   // UNICODE_TO_GBK[27326] := 16#8092;
   // UNICODE_TO_GBK[27327] := 16#C34B;
   // UNICODE_TO_GBK[27328] := 16#8093;
   // UNICODE_TO_GBK[27329] := 16#EBC1;
   // UNICODE_TO_GBK[27330] := 16#8094;
   // UNICODE_TO_GBK[27331] := 16#C34C;
   // UNICODE_TO_GBK[27332] := 16#8095;
   // UNICODE_TO_GBK[27333] := 16#C34D;
   // UNICODE_TO_GBK[27334] := 16#8096;
   // UNICODE_TO_GBK[27335] := 16#D0A4;
   // UNICODE_TO_GBK[27336] := 16#8097;
   // UNICODE_TO_GBK[27337] := 16#C34E;
   // UNICODE_TO_GBK[27338] := 16#8098;
   // UNICODE_TO_GBK[27339] := 16#D6E2;
   // UNICODE_TO_GBK[27340] := 16#8099;
   // UNICODE_TO_GBK[27341] := 16#C34F;
   // UNICODE_TO_GBK[27342] := 16#809A;
   // UNICODE_TO_GBK[27343] := 16#B6C7;
   // UNICODE_TO_GBK[27344] := 16#809B;
   // UNICODE_TO_GBK[27345] := 16#B8D8;
   // UNICODE_TO_GBK[27346] := 16#809C;
   // UNICODE_TO_GBK[27347] := 16#EBC0;
   // UNICODE_TO_GBK[27348] := 16#809D;
   // UNICODE_TO_GBK[27349] := 16#B8CE;
   // UNICODE_TO_GBK[27350] := 16#809E;
   // UNICODE_TO_GBK[27351] := 16#C350;
   // UNICODE_TO_GBK[27352] := 16#809F;
   // UNICODE_TO_GBK[27353] := 16#EBBF;
   // UNICODE_TO_GBK[27354] := 16#80A0;
   // UNICODE_TO_GBK[27355] := 16#B3A6;
   // UNICODE_TO_GBK[27356] := 16#80A1;
   // UNICODE_TO_GBK[27357] := 16#B9C9;
   // UNICODE_TO_GBK[27358] := 16#80A2;
   // UNICODE_TO_GBK[27359] := 16#D6AB;
   // UNICODE_TO_GBK[27360] := 16#80A3;
   // UNICODE_TO_GBK[27361] := 16#C351;
   // UNICODE_TO_GBK[27362] := 16#80A4;
   // UNICODE_TO_GBK[27363] := 16#B7F4;
   // UNICODE_TO_GBK[27364] := 16#80A5;
   // UNICODE_TO_GBK[27365] := 16#B7CA;
   // UNICODE_TO_GBK[27366] := 16#80A6;
   // UNICODE_TO_GBK[27367] := 16#C352;
   // UNICODE_TO_GBK[27368] := 16#80A7;
   // UNICODE_TO_GBK[27369] := 16#C353;
   // UNICODE_TO_GBK[27370] := 16#80A8;
   // UNICODE_TO_GBK[27371] := 16#C354;
   // UNICODE_TO_GBK[27372] := 16#80A9;
   // UNICODE_TO_GBK[27373] := 16#BCE7;
   // UNICODE_TO_GBK[27374] := 16#80AA;
   // UNICODE_TO_GBK[27375] := 16#B7BE;
   // UNICODE_TO_GBK[27376] := 16#80AB;
   // UNICODE_TO_GBK[27377] := 16#EBC6;
   // UNICODE_TO_GBK[27378] := 16#80AC;
   // UNICODE_TO_GBK[27379] := 16#C355;
   // UNICODE_TO_GBK[27380] := 16#80AD;
   // UNICODE_TO_GBK[27381] := 16#EBC7;
   // UNICODE_TO_GBK[27382] := 16#80AE;
   // UNICODE_TO_GBK[27383] := 16#B0B9;
   // UNICODE_TO_GBK[27384] := 16#80AF;
   // UNICODE_TO_GBK[27385] := 16#BFCF;
   // UNICODE_TO_GBK[27386] := 16#80B0;
   // UNICODE_TO_GBK[27387] := 16#C356;
   // UNICODE_TO_GBK[27388] := 16#80B1;
   // UNICODE_TO_GBK[27389] := 16#EBC5;
   // UNICODE_TO_GBK[27390] := 16#80B2;
   // UNICODE_TO_GBK[27391] := 16#D3FD;
   // UNICODE_TO_GBK[27392] := 16#80B3;
   // UNICODE_TO_GBK[27393] := 16#C357;
   // UNICODE_TO_GBK[27394] := 16#80B4;
   // UNICODE_TO_GBK[27395] := 16#EBC8;
   // UNICODE_TO_GBK[27396] := 16#80B5;
   // UNICODE_TO_GBK[27397] := 16#C358;
   // UNICODE_TO_GBK[27398] := 16#80B6;
   // UNICODE_TO_GBK[27399] := 16#C359;
   // UNICODE_TO_GBK[27400] := 16#80B7;
   // UNICODE_TO_GBK[27401] := 16#EBC9;
   // UNICODE_TO_GBK[27402] := 16#80B8;
   // UNICODE_TO_GBK[27403] := 16#C35A;
   // UNICODE_TO_GBK[27404] := 16#80B9;
   // UNICODE_TO_GBK[27405] := 16#C35B;
   // UNICODE_TO_GBK[27406] := 16#80BA;
   // UNICODE_TO_GBK[27407] := 16#B7CE;
   // UNICODE_TO_GBK[27408] := 16#80BB;
   // UNICODE_TO_GBK[27409] := 16#C35C;
   // UNICODE_TO_GBK[27410] := 16#80BC;
   // UNICODE_TO_GBK[27411] := 16#EBC2;
   // UNICODE_TO_GBK[27412] := 16#80BD;
   // UNICODE_TO_GBK[27413] := 16#EBC4;
   // UNICODE_TO_GBK[27414] := 16#80BE;
   // UNICODE_TO_GBK[27415] := 16#C9F6;
   // UNICODE_TO_GBK[27416] := 16#80BF;
   // UNICODE_TO_GBK[27417] := 16#D6D7;
   // UNICODE_TO_GBK[27418] := 16#80C0;
   // UNICODE_TO_GBK[27419] := 16#D5CD;
   // UNICODE_TO_GBK[27420] := 16#80C1;
   // UNICODE_TO_GBK[27421] := 16#D0B2;
   // UNICODE_TO_GBK[27422] := 16#80C2;
   // UNICODE_TO_GBK[27423] := 16#EBCF;
   // UNICODE_TO_GBK[27424] := 16#80C3;
   // UNICODE_TO_GBK[27425] := 16#CEB8;
   // UNICODE_TO_GBK[27426] := 16#80C4;
   // UNICODE_TO_GBK[27427] := 16#EBD0;
   // UNICODE_TO_GBK[27428] := 16#80C5;
   // UNICODE_TO_GBK[27429] := 16#C35D;
   // UNICODE_TO_GBK[27430] := 16#80C6;
   // UNICODE_TO_GBK[27431] := 16#B5A8;
   // UNICODE_TO_GBK[27432] := 16#80C7;
   // UNICODE_TO_GBK[27433] := 16#C35E;
   // UNICODE_TO_GBK[27434] := 16#80C8;
   // UNICODE_TO_GBK[27435] := 16#C35F;
   // UNICODE_TO_GBK[27436] := 16#80C9;
   // UNICODE_TO_GBK[27437] := 16#C360;
   // UNICODE_TO_GBK[27438] := 16#80CA;
   // UNICODE_TO_GBK[27439] := 16#C361;
   // UNICODE_TO_GBK[27440] := 16#80CB;
   // UNICODE_TO_GBK[27441] := 16#C362;
   // UNICODE_TO_GBK[27442] := 16#80CC;
   // UNICODE_TO_GBK[27443] := 16#B1B3;
   // UNICODE_TO_GBK[27444] := 16#80CD;
   // UNICODE_TO_GBK[27445] := 16#EBD2;
   // UNICODE_TO_GBK[27446] := 16#80CE;
   // UNICODE_TO_GBK[27447] := 16#CCA5;
   // UNICODE_TO_GBK[27448] := 16#80CF;
   // UNICODE_TO_GBK[27449] := 16#C363;
   // UNICODE_TO_GBK[27450] := 16#80D0;
   // UNICODE_TO_GBK[27451] := 16#C364;
   // UNICODE_TO_GBK[27452] := 16#80D1;
   // UNICODE_TO_GBK[27453] := 16#C365;
   // UNICODE_TO_GBK[27454] := 16#80D2;
   // UNICODE_TO_GBK[27455] := 16#C366;
   // UNICODE_TO_GBK[27456] := 16#80D3;
   // UNICODE_TO_GBK[27457] := 16#C367;
   // UNICODE_TO_GBK[27458] := 16#80D4;
   // UNICODE_TO_GBK[27459] := 16#C368;
   // UNICODE_TO_GBK[27460] := 16#80D5;
   // UNICODE_TO_GBK[27461] := 16#C369;
   // UNICODE_TO_GBK[27462] := 16#80D6;
   // UNICODE_TO_GBK[27463] := 16#C5D6;
   // UNICODE_TO_GBK[27464] := 16#80D7;
   // UNICODE_TO_GBK[27465] := 16#EBD3;
   // UNICODE_TO_GBK[27466] := 16#80D8;
   // UNICODE_TO_GBK[27467] := 16#C36A;
   // UNICODE_TO_GBK[27468] := 16#80D9;
   // UNICODE_TO_GBK[27469] := 16#EBD1;
   // UNICODE_TO_GBK[27470] := 16#80DA;
   // UNICODE_TO_GBK[27471] := 16#C5DF;
   // UNICODE_TO_GBK[27472] := 16#80DB;
   // UNICODE_TO_GBK[27473] := 16#EBCE;
   // UNICODE_TO_GBK[27474] := 16#80DC;
   // UNICODE_TO_GBK[27475] := 16#CAA4;
   // UNICODE_TO_GBK[27476] := 16#80DD;
   // UNICODE_TO_GBK[27477] := 16#EBD5;
   // UNICODE_TO_GBK[27478] := 16#80DE;
   // UNICODE_TO_GBK[27479] := 16#B0FB;
   // UNICODE_TO_GBK[27480] := 16#80DF;
   // UNICODE_TO_GBK[27481] := 16#C36B;
   // UNICODE_TO_GBK[27482] := 16#80E0;
   // UNICODE_TO_GBK[27483] := 16#C36C;
   // UNICODE_TO_GBK[27484] := 16#80E1;
   // UNICODE_TO_GBK[27485] := 16#BAFA;
   // UNICODE_TO_GBK[27486] := 16#80E2;
   // UNICODE_TO_GBK[27487] := 16#C36D;
   // UNICODE_TO_GBK[27488] := 16#80E3;
   // UNICODE_TO_GBK[27489] := 16#C36E;
   // UNICODE_TO_GBK[27490] := 16#80E4;
   // UNICODE_TO_GBK[27491] := 16#D8B7;
   // UNICODE_TO_GBK[27492] := 16#80E5;
   // UNICODE_TO_GBK[27493] := 16#F1E3;
   // UNICODE_TO_GBK[27494] := 16#80E6;
   // UNICODE_TO_GBK[27495] := 16#C36F;
   // UNICODE_TO_GBK[27496] := 16#80E7;
   // UNICODE_TO_GBK[27497] := 16#EBCA;
   // UNICODE_TO_GBK[27498] := 16#80E8;
   // UNICODE_TO_GBK[27499] := 16#EBCB;
   // UNICODE_TO_GBK[27500] := 16#80E9;
   // UNICODE_TO_GBK[27501] := 16#EBCC;
   // UNICODE_TO_GBK[27502] := 16#80EA;
   // UNICODE_TO_GBK[27503] := 16#EBCD;
   // UNICODE_TO_GBK[27504] := 16#80EB;
   // UNICODE_TO_GBK[27505] := 16#EBD6;
   // UNICODE_TO_GBK[27506] := 16#80EC;
   // UNICODE_TO_GBK[27507] := 16#E6C0;
   // UNICODE_TO_GBK[27508] := 16#80ED;
   // UNICODE_TO_GBK[27509] := 16#EBD9;
   // UNICODE_TO_GBK[27510] := 16#80EE;
   // UNICODE_TO_GBK[27511] := 16#C370;
   // UNICODE_TO_GBK[27512] := 16#80EF;
   // UNICODE_TO_GBK[27513] := 16#BFE8;
   // UNICODE_TO_GBK[27514] := 16#80F0;
   // UNICODE_TO_GBK[27515] := 16#D2C8;
   // UNICODE_TO_GBK[27516] := 16#80F1;
   // UNICODE_TO_GBK[27517] := 16#EBD7;
   // UNICODE_TO_GBK[27518] := 16#80F2;
   // UNICODE_TO_GBK[27519] := 16#EBDC;
   // UNICODE_TO_GBK[27520] := 16#80F3;
   // UNICODE_TO_GBK[27521] := 16#B8EC;
   // UNICODE_TO_GBK[27522] := 16#80F4;
   // UNICODE_TO_GBK[27523] := 16#EBD8;
   // UNICODE_TO_GBK[27524] := 16#80F5;
   // UNICODE_TO_GBK[27525] := 16#C371;
   // UNICODE_TO_GBK[27526] := 16#80F6;
   // UNICODE_TO_GBK[27527] := 16#BDBA;
   // UNICODE_TO_GBK[27528] := 16#80F7;
   // UNICODE_TO_GBK[27529] := 16#C372;
   // UNICODE_TO_GBK[27530] := 16#80F8;
   // UNICODE_TO_GBK[27531] := 16#D0D8;
   // UNICODE_TO_GBK[27532] := 16#80F9;
   // UNICODE_TO_GBK[27533] := 16#C373;
   // UNICODE_TO_GBK[27534] := 16#80FA;
   // UNICODE_TO_GBK[27535] := 16#B0B7;
   // UNICODE_TO_GBK[27536] := 16#80FB;
   // UNICODE_TO_GBK[27537] := 16#C374;
   // UNICODE_TO_GBK[27538] := 16#80FC;
   // UNICODE_TO_GBK[27539] := 16#EBDD;
   // UNICODE_TO_GBK[27540] := 16#80FD;
   // UNICODE_TO_GBK[27541] := 16#C4DC;
   // UNICODE_TO_GBK[27542] := 16#80FE;
   // UNICODE_TO_GBK[27543] := 16#C375;
   // UNICODE_TO_GBK[27544] := 16#80FF;
   // UNICODE_TO_GBK[27545] := 16#C376;
   // UNICODE_TO_GBK[27546] := 16#8100;
   // UNICODE_TO_GBK[27547] := 16#C377;
   // UNICODE_TO_GBK[27548] := 16#8101;
   // UNICODE_TO_GBK[27549] := 16#C378;
   // UNICODE_TO_GBK[27550] := 16#8102;
   // UNICODE_TO_GBK[27551] := 16#D6AC;
   // UNICODE_TO_GBK[27552] := 16#8103;
   // UNICODE_TO_GBK[27553] := 16#C379;
   // UNICODE_TO_GBK[27554] := 16#8104;
   // UNICODE_TO_GBK[27555] := 16#C37A;
   // UNICODE_TO_GBK[27556] := 16#8105;
   // UNICODE_TO_GBK[27557] := 16#C37B;
   // UNICODE_TO_GBK[27558] := 16#8106;
   // UNICODE_TO_GBK[27559] := 16#B4E0;
   // UNICODE_TO_GBK[27560] := 16#8107;
   // UNICODE_TO_GBK[27561] := 16#C37C;
   // UNICODE_TO_GBK[27562] := 16#8108;
   // UNICODE_TO_GBK[27563] := 16#C37D;
   // UNICODE_TO_GBK[27564] := 16#8109;
   // UNICODE_TO_GBK[27565] := 16#C2F6;
   // UNICODE_TO_GBK[27566] := 16#810A;
   // UNICODE_TO_GBK[27567] := 16#BCB9;
   // UNICODE_TO_GBK[27568] := 16#810B;
   // UNICODE_TO_GBK[27569] := 16#C37E;
   // UNICODE_TO_GBK[27570] := 16#810C;
   // UNICODE_TO_GBK[27571] := 16#C380;
   // UNICODE_TO_GBK[27572] := 16#810D;
   // UNICODE_TO_GBK[27573] := 16#EBDA;
   // UNICODE_TO_GBK[27574] := 16#810E;
   // UNICODE_TO_GBK[27575] := 16#EBDB;
   // UNICODE_TO_GBK[27576] := 16#810F;
   // UNICODE_TO_GBK[27577] := 16#D4E0;
   // UNICODE_TO_GBK[27578] := 16#8110;
   // UNICODE_TO_GBK[27579] := 16#C6EA;
   // UNICODE_TO_GBK[27580] := 16#8111;
   // UNICODE_TO_GBK[27581] := 16#C4D4;
   // UNICODE_TO_GBK[27582] := 16#8112;
   // UNICODE_TO_GBK[27583] := 16#EBDF;
   // UNICODE_TO_GBK[27584] := 16#8113;
   // UNICODE_TO_GBK[27585] := 16#C5A7;
   // UNICODE_TO_GBK[27586] := 16#8114;
   // UNICODE_TO_GBK[27587] := 16#D9F5;
   // UNICODE_TO_GBK[27588] := 16#8115;
   // UNICODE_TO_GBK[27589] := 16#C381;
   // UNICODE_TO_GBK[27590] := 16#8116;
   // UNICODE_TO_GBK[27591] := 16#B2B1;
   // UNICODE_TO_GBK[27592] := 16#8117;
   // UNICODE_TO_GBK[27593] := 16#C382;
   // UNICODE_TO_GBK[27594] := 16#8118;
   // UNICODE_TO_GBK[27595] := 16#EBE4;
   // UNICODE_TO_GBK[27596] := 16#8119;
   // UNICODE_TO_GBK[27597] := 16#C383;
   // UNICODE_TO_GBK[27598] := 16#811A;
   // UNICODE_TO_GBK[27599] := 16#BDC5;
   // UNICODE_TO_GBK[27600] := 16#811B;
   // UNICODE_TO_GBK[27601] := 16#C384;
   // UNICODE_TO_GBK[27602] := 16#811C;
   // UNICODE_TO_GBK[27603] := 16#C385;
   // UNICODE_TO_GBK[27604] := 16#811D;
   // UNICODE_TO_GBK[27605] := 16#C386;
   // UNICODE_TO_GBK[27606] := 16#811E;
   // UNICODE_TO_GBK[27607] := 16#EBE2;
   // UNICODE_TO_GBK[27608] := 16#811F;
   // UNICODE_TO_GBK[27609] := 16#C387;
   // UNICODE_TO_GBK[27610] := 16#8120;
   // UNICODE_TO_GBK[27611] := 16#C388;
   // UNICODE_TO_GBK[27612] := 16#8121;
   // UNICODE_TO_GBK[27613] := 16#C389;
   // UNICODE_TO_GBK[27614] := 16#8122;
   // UNICODE_TO_GBK[27615] := 16#C38A;
   // UNICODE_TO_GBK[27616] := 16#8123;
   // UNICODE_TO_GBK[27617] := 16#C38B;
   // UNICODE_TO_GBK[27618] := 16#8124;
   // UNICODE_TO_GBK[27619] := 16#C38C;
   // UNICODE_TO_GBK[27620] := 16#8125;
   // UNICODE_TO_GBK[27621] := 16#C38D;
   // UNICODE_TO_GBK[27622] := 16#8126;
   // UNICODE_TO_GBK[27623] := 16#C38E;
   // UNICODE_TO_GBK[27624] := 16#8127;
   // UNICODE_TO_GBK[27625] := 16#C38F;
   // UNICODE_TO_GBK[27626] := 16#8128;
   // UNICODE_TO_GBK[27627] := 16#C390;
   // UNICODE_TO_GBK[27628] := 16#8129;
   // UNICODE_TO_GBK[27629] := 16#C391;
   // UNICODE_TO_GBK[27630] := 16#812A;
   // UNICODE_TO_GBK[27631] := 16#C392;
   // UNICODE_TO_GBK[27632] := 16#812B;
   // UNICODE_TO_GBK[27633] := 16#C393;
   // UNICODE_TO_GBK[27634] := 16#812C;
   // UNICODE_TO_GBK[27635] := 16#EBE3;
   // UNICODE_TO_GBK[27636] := 16#812D;
   // UNICODE_TO_GBK[27637] := 16#C394;
   // UNICODE_TO_GBK[27638] := 16#812E;
   // UNICODE_TO_GBK[27639] := 16#C395;
   // UNICODE_TO_GBK[27640] := 16#812F;
   // UNICODE_TO_GBK[27641] := 16#B8AC;
   // UNICODE_TO_GBK[27642] := 16#8130;
   // UNICODE_TO_GBK[27643] := 16#C396;
   // UNICODE_TO_GBK[27644] := 16#8131;
   // UNICODE_TO_GBK[27645] := 16#CDD1;
   // UNICODE_TO_GBK[27646] := 16#8132;
   // UNICODE_TO_GBK[27647] := 16#EBE5;
   // UNICODE_TO_GBK[27648] := 16#8133;
   // UNICODE_TO_GBK[27649] := 16#C397;
   // UNICODE_TO_GBK[27650] := 16#8134;
   // UNICODE_TO_GBK[27651] := 16#C398;
   // UNICODE_TO_GBK[27652] := 16#8135;
   // UNICODE_TO_GBK[27653] := 16#C399;
   // UNICODE_TO_GBK[27654] := 16#8136;
   // UNICODE_TO_GBK[27655] := 16#EBE1;
   // UNICODE_TO_GBK[27656] := 16#8137;
   // UNICODE_TO_GBK[27657] := 16#C39A;
   // UNICODE_TO_GBK[27658] := 16#8138;
   // UNICODE_TO_GBK[27659] := 16#C1B3;
   // UNICODE_TO_GBK[27660] := 16#8139;
   // UNICODE_TO_GBK[27661] := 16#C39B;
   // UNICODE_TO_GBK[27662] := 16#813A;
   // UNICODE_TO_GBK[27663] := 16#C39C;
   // UNICODE_TO_GBK[27664] := 16#813B;
   // UNICODE_TO_GBK[27665] := 16#C39D;
   // UNICODE_TO_GBK[27666] := 16#813C;
   // UNICODE_TO_GBK[27667] := 16#C39E;
   // UNICODE_TO_GBK[27668] := 16#813D;
   // UNICODE_TO_GBK[27669] := 16#C39F;
   // UNICODE_TO_GBK[27670] := 16#813E;
   // UNICODE_TO_GBK[27671] := 16#C6A2;
   // UNICODE_TO_GBK[27672] := 16#813F;
   // UNICODE_TO_GBK[27673] := 16#C3A0;
   // UNICODE_TO_GBK[27674] := 16#8140;
   // UNICODE_TO_GBK[27675] := 16#C440;
   // UNICODE_TO_GBK[27676] := 16#8141;
   // UNICODE_TO_GBK[27677] := 16#C441;
   // UNICODE_TO_GBK[27678] := 16#8142;
   // UNICODE_TO_GBK[27679] := 16#C442;
   // UNICODE_TO_GBK[27680] := 16#8143;
   // UNICODE_TO_GBK[27681] := 16#C443;
   // UNICODE_TO_GBK[27682] := 16#8144;
   // UNICODE_TO_GBK[27683] := 16#C444;
   // UNICODE_TO_GBK[27684] := 16#8145;
   // UNICODE_TO_GBK[27685] := 16#C445;
   // UNICODE_TO_GBK[27686] := 16#8146;
   // UNICODE_TO_GBK[27687] := 16#CCF3;
   // UNICODE_TO_GBK[27688] := 16#8147;
   // UNICODE_TO_GBK[27689] := 16#C446;
   // UNICODE_TO_GBK[27690] := 16#8148;
   // UNICODE_TO_GBK[27691] := 16#EBE6;
   // UNICODE_TO_GBK[27692] := 16#8149;
   // UNICODE_TO_GBK[27693] := 16#C447;
   // UNICODE_TO_GBK[27694] := 16#814A;
   // UNICODE_TO_GBK[27695] := 16#C0B0;
   // UNICODE_TO_GBK[27696] := 16#814B;
   // UNICODE_TO_GBK[27697] := 16#D2B8;
   // UNICODE_TO_GBK[27698] := 16#814C;
   // UNICODE_TO_GBK[27699] := 16#EBE7;
   // UNICODE_TO_GBK[27700] := 16#814D;
   // UNICODE_TO_GBK[27701] := 16#C448;
   // UNICODE_TO_GBK[27702] := 16#814E;
   // UNICODE_TO_GBK[27703] := 16#C449;
   // UNICODE_TO_GBK[27704] := 16#814F;
   // UNICODE_TO_GBK[27705] := 16#C44A;
   // UNICODE_TO_GBK[27706] := 16#8150;
   // UNICODE_TO_GBK[27707] := 16#B8AF;
   // UNICODE_TO_GBK[27708] := 16#8151;
   // UNICODE_TO_GBK[27709] := 16#B8AD;
   // UNICODE_TO_GBK[27710] := 16#8152;
   // UNICODE_TO_GBK[27711] := 16#C44B;
   // UNICODE_TO_GBK[27712] := 16#8153;
   // UNICODE_TO_GBK[27713] := 16#EBE8;
   // UNICODE_TO_GBK[27714] := 16#8154;
   // UNICODE_TO_GBK[27715] := 16#C7BB;
   // UNICODE_TO_GBK[27716] := 16#8155;
   // UNICODE_TO_GBK[27717] := 16#CDF3;
   // UNICODE_TO_GBK[27718] := 16#8156;
   // UNICODE_TO_GBK[27719] := 16#C44C;
   // UNICODE_TO_GBK[27720] := 16#8157;
   // UNICODE_TO_GBK[27721] := 16#C44D;
   // UNICODE_TO_GBK[27722] := 16#8158;
   // UNICODE_TO_GBK[27723] := 16#C44E;
   // UNICODE_TO_GBK[27724] := 16#8159;
   // UNICODE_TO_GBK[27725] := 16#EBEA;
   // UNICODE_TO_GBK[27726] := 16#815A;
   // UNICODE_TO_GBK[27727] := 16#EBEB;
   // UNICODE_TO_GBK[27728] := 16#815B;
   // UNICODE_TO_GBK[27729] := 16#C44F;
   // UNICODE_TO_GBK[27730] := 16#815C;
   // UNICODE_TO_GBK[27731] := 16#C450;
   // UNICODE_TO_GBK[27732] := 16#815D;
   // UNICODE_TO_GBK[27733] := 16#C451;
   // UNICODE_TO_GBK[27734] := 16#815E;
   // UNICODE_TO_GBK[27735] := 16#C452;
   // UNICODE_TO_GBK[27736] := 16#815F;
   // UNICODE_TO_GBK[27737] := 16#C453;
   // UNICODE_TO_GBK[27738] := 16#8160;
   // UNICODE_TO_GBK[27739] := 16#EBED;
   // UNICODE_TO_GBK[27740] := 16#8161;
   // UNICODE_TO_GBK[27741] := 16#C454;
   // UNICODE_TO_GBK[27742] := 16#8162;
   // UNICODE_TO_GBK[27743] := 16#C455;
   // UNICODE_TO_GBK[27744] := 16#8163;
   // UNICODE_TO_GBK[27745] := 16#C456;
   // UNICODE_TO_GBK[27746] := 16#8164;
   // UNICODE_TO_GBK[27747] := 16#C457;
   // UNICODE_TO_GBK[27748] := 16#8165;
   // UNICODE_TO_GBK[27749] := 16#D0C8;
   // UNICODE_TO_GBK[27750] := 16#8166;
   // UNICODE_TO_GBK[27751] := 16#C458;
   // UNICODE_TO_GBK[27752] := 16#8167;
   // UNICODE_TO_GBK[27753] := 16#EBF2;
   // UNICODE_TO_GBK[27754] := 16#8168;
   // UNICODE_TO_GBK[27755] := 16#C459;
   // UNICODE_TO_GBK[27756] := 16#8169;
   // UNICODE_TO_GBK[27757] := 16#EBEE;
   // UNICODE_TO_GBK[27758] := 16#816A;
   // UNICODE_TO_GBK[27759] := 16#C45A;
   // UNICODE_TO_GBK[27760] := 16#816B;
   // UNICODE_TO_GBK[27761] := 16#C45B;
   // UNICODE_TO_GBK[27762] := 16#816C;
   // UNICODE_TO_GBK[27763] := 16#C45C;
   // UNICODE_TO_GBK[27764] := 16#816D;
   // UNICODE_TO_GBK[27765] := 16#EBF1;
   // UNICODE_TO_GBK[27766] := 16#816E;
   // UNICODE_TO_GBK[27767] := 16#C8F9;
   // UNICODE_TO_GBK[27768] := 16#816F;
   // UNICODE_TO_GBK[27769] := 16#C45D;
   // UNICODE_TO_GBK[27770] := 16#8170;
   // UNICODE_TO_GBK[27771] := 16#D1FC;
   // UNICODE_TO_GBK[27772] := 16#8171;
   // UNICODE_TO_GBK[27773] := 16#EBEC;
   // UNICODE_TO_GBK[27774] := 16#8172;
   // UNICODE_TO_GBK[27775] := 16#C45E;
   // UNICODE_TO_GBK[27776] := 16#8173;
   // UNICODE_TO_GBK[27777] := 16#C45F;
   // UNICODE_TO_GBK[27778] := 16#8174;
   // UNICODE_TO_GBK[27779] := 16#EBE9;
   // UNICODE_TO_GBK[27780] := 16#8175;
   // UNICODE_TO_GBK[27781] := 16#C460;
   // UNICODE_TO_GBK[27782] := 16#8176;
   // UNICODE_TO_GBK[27783] := 16#C461;
   // UNICODE_TO_GBK[27784] := 16#8177;
   // UNICODE_TO_GBK[27785] := 16#C462;
   // UNICODE_TO_GBK[27786] := 16#8178;
   // UNICODE_TO_GBK[27787] := 16#C463;
   // UNICODE_TO_GBK[27788] := 16#8179;
   // UNICODE_TO_GBK[27789] := 16#B8B9;
   // UNICODE_TO_GBK[27790] := 16#817A;
   // UNICODE_TO_GBK[27791] := 16#CFD9;
   // UNICODE_TO_GBK[27792] := 16#817B;
   // UNICODE_TO_GBK[27793] := 16#C4E5;
   // UNICODE_TO_GBK[27794] := 16#817C;
   // UNICODE_TO_GBK[27795] := 16#EBEF;
   // UNICODE_TO_GBK[27796] := 16#817D;
   // UNICODE_TO_GBK[27797] := 16#EBF0;
   // UNICODE_TO_GBK[27798] := 16#817E;
   // UNICODE_TO_GBK[27799] := 16#CCDA;
   // UNICODE_TO_GBK[27800] := 16#817F;
   // UNICODE_TO_GBK[27801] := 16#CDC8;
   // UNICODE_TO_GBK[27802] := 16#8180;
   // UNICODE_TO_GBK[27803] := 16#B0F2;
   // UNICODE_TO_GBK[27804] := 16#8181;
   // UNICODE_TO_GBK[27805] := 16#C464;
   // UNICODE_TO_GBK[27806] := 16#8182;
   // UNICODE_TO_GBK[27807] := 16#EBF6;
   // UNICODE_TO_GBK[27808] := 16#8183;
   // UNICODE_TO_GBK[27809] := 16#C465;
   // UNICODE_TO_GBK[27810] := 16#8184;
   // UNICODE_TO_GBK[27811] := 16#C466;
   // UNICODE_TO_GBK[27812] := 16#8185;
   // UNICODE_TO_GBK[27813] := 16#C467;
   // UNICODE_TO_GBK[27814] := 16#8186;
   // UNICODE_TO_GBK[27815] := 16#C468;
   // UNICODE_TO_GBK[27816] := 16#8187;
   // UNICODE_TO_GBK[27817] := 16#C469;
   // UNICODE_TO_GBK[27818] := 16#8188;
   // UNICODE_TO_GBK[27819] := 16#EBF5;
   // UNICODE_TO_GBK[27820] := 16#8189;
   // UNICODE_TO_GBK[27821] := 16#C46A;
   // UNICODE_TO_GBK[27822] := 16#818A;
   // UNICODE_TO_GBK[27823] := 16#B2B2;
   // UNICODE_TO_GBK[27824] := 16#818B;
   // UNICODE_TO_GBK[27825] := 16#C46B;
   // UNICODE_TO_GBK[27826] := 16#818C;
   // UNICODE_TO_GBK[27827] := 16#C46C;
   // UNICODE_TO_GBK[27828] := 16#818D;
   // UNICODE_TO_GBK[27829] := 16#C46D;
   // UNICODE_TO_GBK[27830] := 16#818E;
   // UNICODE_TO_GBK[27831] := 16#C46E;
   // UNICODE_TO_GBK[27832] := 16#818F;
   // UNICODE_TO_GBK[27833] := 16#B8E0;
   // UNICODE_TO_GBK[27834] := 16#8190;
   // UNICODE_TO_GBK[27835] := 16#C46F;
   // UNICODE_TO_GBK[27836] := 16#8191;
   // UNICODE_TO_GBK[27837] := 16#EBF7;
   // UNICODE_TO_GBK[27838] := 16#8192;
   // UNICODE_TO_GBK[27839] := 16#C470;
   // UNICODE_TO_GBK[27840] := 16#8193;
   // UNICODE_TO_GBK[27841] := 16#C471;
   // UNICODE_TO_GBK[27842] := 16#8194;
   // UNICODE_TO_GBK[27843] := 16#C472;
   // UNICODE_TO_GBK[27844] := 16#8195;
   // UNICODE_TO_GBK[27845] := 16#C473;
   // UNICODE_TO_GBK[27846] := 16#8196;
   // UNICODE_TO_GBK[27847] := 16#C474;
   // UNICODE_TO_GBK[27848] := 16#8197;
   // UNICODE_TO_GBK[27849] := 16#C475;
   // UNICODE_TO_GBK[27850] := 16#8198;
   // UNICODE_TO_GBK[27851] := 16#B1EC;
   // UNICODE_TO_GBK[27852] := 16#8199;
   // UNICODE_TO_GBK[27853] := 16#C476;
   // UNICODE_TO_GBK[27854] := 16#819A;
   // UNICODE_TO_GBK[27855] := 16#C477;
   // UNICODE_TO_GBK[27856] := 16#819B;
   // UNICODE_TO_GBK[27857] := 16#CCC5;
   // UNICODE_TO_GBK[27858] := 16#819C;
   // UNICODE_TO_GBK[27859] := 16#C4A4;
   // UNICODE_TO_GBK[27860] := 16#819D;
   // UNICODE_TO_GBK[27861] := 16#CFA5;
   // UNICODE_TO_GBK[27862] := 16#819E;
   // UNICODE_TO_GBK[27863] := 16#C478;
   // UNICODE_TO_GBK[27864] := 16#819F;
   // UNICODE_TO_GBK[27865] := 16#C479;
   // UNICODE_TO_GBK[27866] := 16#81A0;
   // UNICODE_TO_GBK[27867] := 16#C47A;
   // UNICODE_TO_GBK[27868] := 16#81A1;
   // UNICODE_TO_GBK[27869] := 16#C47B;
   // UNICODE_TO_GBK[27870] := 16#81A2;
   // UNICODE_TO_GBK[27871] := 16#C47C;
   // UNICODE_TO_GBK[27872] := 16#81A3;
   // UNICODE_TO_GBK[27873] := 16#EBF9;
   // UNICODE_TO_GBK[27874] := 16#81A4;
   // UNICODE_TO_GBK[27875] := 16#C47D;
   // UNICODE_TO_GBK[27876] := 16#81A5;
   // UNICODE_TO_GBK[27877] := 16#C47E;
   // UNICODE_TO_GBK[27878] := 16#81A6;
   // UNICODE_TO_GBK[27879] := 16#ECA2;
   // UNICODE_TO_GBK[27880] := 16#81A7;
   // UNICODE_TO_GBK[27881] := 16#C480;
   // UNICODE_TO_GBK[27882] := 16#81A8;
   // UNICODE_TO_GBK[27883] := 16#C5F2;
   // UNICODE_TO_GBK[27884] := 16#81A9;
   // UNICODE_TO_GBK[27885] := 16#C481;
   // UNICODE_TO_GBK[27886] := 16#81AA;
   // UNICODE_TO_GBK[27887] := 16#EBFA;
   // UNICODE_TO_GBK[27888] := 16#81AB;
   // UNICODE_TO_GBK[27889] := 16#C482;
   // UNICODE_TO_GBK[27890] := 16#81AC;
   // UNICODE_TO_GBK[27891] := 16#C483;
   // UNICODE_TO_GBK[27892] := 16#81AD;
   // UNICODE_TO_GBK[27893] := 16#C484;
   // UNICODE_TO_GBK[27894] := 16#81AE;
   // UNICODE_TO_GBK[27895] := 16#C485;
   // UNICODE_TO_GBK[27896] := 16#81AF;
   // UNICODE_TO_GBK[27897] := 16#C486;
   // UNICODE_TO_GBK[27898] := 16#81B0;
   // UNICODE_TO_GBK[27899] := 16#C487;
   // UNICODE_TO_GBK[27900] := 16#81B1;
   // UNICODE_TO_GBK[27901] := 16#C488;
   // UNICODE_TO_GBK[27902] := 16#81B2;
   // UNICODE_TO_GBK[27903] := 16#C489;
   // UNICODE_TO_GBK[27904] := 16#81B3;
   // UNICODE_TO_GBK[27905] := 16#C9C5;
   // UNICODE_TO_GBK[27906] := 16#81B4;
   // UNICODE_TO_GBK[27907] := 16#C48A;
   // UNICODE_TO_GBK[27908] := 16#81B5;
   // UNICODE_TO_GBK[27909] := 16#C48B;
   // UNICODE_TO_GBK[27910] := 16#81B6;
   // UNICODE_TO_GBK[27911] := 16#C48C;
   // UNICODE_TO_GBK[27912] := 16#81B7;
   // UNICODE_TO_GBK[27913] := 16#C48D;
   // UNICODE_TO_GBK[27914] := 16#81B8;
   // UNICODE_TO_GBK[27915] := 16#C48E;
   // UNICODE_TO_GBK[27916] := 16#81B9;
   // UNICODE_TO_GBK[27917] := 16#C48F;
   // UNICODE_TO_GBK[27918] := 16#81BA;
   // UNICODE_TO_GBK[27919] := 16#E2DF;
   // UNICODE_TO_GBK[27920] := 16#81BB;
   // UNICODE_TO_GBK[27921] := 16#EBFE;
   // UNICODE_TO_GBK[27922] := 16#81BC;
   // UNICODE_TO_GBK[27923] := 16#C490;
   // UNICODE_TO_GBK[27924] := 16#81BD;
   // UNICODE_TO_GBK[27925] := 16#C491;
   // UNICODE_TO_GBK[27926] := 16#81BE;
   // UNICODE_TO_GBK[27927] := 16#C492;
   // UNICODE_TO_GBK[27928] := 16#81BF;
   // UNICODE_TO_GBK[27929] := 16#C493;
   // UNICODE_TO_GBK[27930] := 16#81C0;
   // UNICODE_TO_GBK[27931] := 16#CDCE;
   // UNICODE_TO_GBK[27932] := 16#81C1;
   // UNICODE_TO_GBK[27933] := 16#ECA1;
   // UNICODE_TO_GBK[27934] := 16#81C2;
   // UNICODE_TO_GBK[27935] := 16#B1DB;
   // UNICODE_TO_GBK[27936] := 16#81C3;
   // UNICODE_TO_GBK[27937] := 16#D3B7;
   // UNICODE_TO_GBK[27938] := 16#81C4;
   // UNICODE_TO_GBK[27939] := 16#C494;
   // UNICODE_TO_GBK[27940] := 16#81C5;
   // UNICODE_TO_GBK[27941] := 16#C495;
   // UNICODE_TO_GBK[27942] := 16#81C6;
   // UNICODE_TO_GBK[27943] := 16#D2DC;
   // UNICODE_TO_GBK[27944] := 16#81C7;
   // UNICODE_TO_GBK[27945] := 16#C496;
   // UNICODE_TO_GBK[27946] := 16#81C8;
   // UNICODE_TO_GBK[27947] := 16#C497;
   // UNICODE_TO_GBK[27948] := 16#81C9;
   // UNICODE_TO_GBK[27949] := 16#C498;
   // UNICODE_TO_GBK[27950] := 16#81CA;
   // UNICODE_TO_GBK[27951] := 16#EBFD;
   // UNICODE_TO_GBK[27952] := 16#81CB;
   // UNICODE_TO_GBK[27953] := 16#C499;
   // UNICODE_TO_GBK[27954] := 16#81CC;
   // UNICODE_TO_GBK[27955] := 16#EBFB;
   // UNICODE_TO_GBK[27956] := 16#81CD;
   // UNICODE_TO_GBK[27957] := 16#C49A;
   // UNICODE_TO_GBK[27958] := 16#81CE;
   // UNICODE_TO_GBK[27959] := 16#C49B;
   // UNICODE_TO_GBK[27960] := 16#81CF;
   // UNICODE_TO_GBK[27961] := 16#C49C;
   // UNICODE_TO_GBK[27962] := 16#81D0;
   // UNICODE_TO_GBK[27963] := 16#C49D;
   // UNICODE_TO_GBK[27964] := 16#81D1;
   // UNICODE_TO_GBK[27965] := 16#C49E;
   // UNICODE_TO_GBK[27966] := 16#81D2;
   // UNICODE_TO_GBK[27967] := 16#C49F;
   // UNICODE_TO_GBK[27968] := 16#81D3;
   // UNICODE_TO_GBK[27969] := 16#C4A0;
   // UNICODE_TO_GBK[27970] := 16#81D4;
   // UNICODE_TO_GBK[27971] := 16#C540;
   // UNICODE_TO_GBK[27972] := 16#81D5;
   // UNICODE_TO_GBK[27973] := 16#C541;
   // UNICODE_TO_GBK[27974] := 16#81D6;
   // UNICODE_TO_GBK[27975] := 16#C542;
   // UNICODE_TO_GBK[27976] := 16#81D7;
   // UNICODE_TO_GBK[27977] := 16#C543;
   // UNICODE_TO_GBK[27978] := 16#81D8;
   // UNICODE_TO_GBK[27979] := 16#C544;
   // UNICODE_TO_GBK[27980] := 16#81D9;
   // UNICODE_TO_GBK[27981] := 16#C545;
   // UNICODE_TO_GBK[27982] := 16#81DA;
   // UNICODE_TO_GBK[27983] := 16#C546;
   // UNICODE_TO_GBK[27984] := 16#81DB;
   // UNICODE_TO_GBK[27985] := 16#C547;
   // UNICODE_TO_GBK[27986] := 16#81DC;
   // UNICODE_TO_GBK[27987] := 16#C548;
   // UNICODE_TO_GBK[27988] := 16#81DD;
   // UNICODE_TO_GBK[27989] := 16#C549;
   // UNICODE_TO_GBK[27990] := 16#81DE;
   // UNICODE_TO_GBK[27991] := 16#C54A;
   // UNICODE_TO_GBK[27992] := 16#81DF;
   // UNICODE_TO_GBK[27993] := 16#C54B;
   // UNICODE_TO_GBK[27994] := 16#81E0;
   // UNICODE_TO_GBK[27995] := 16#C54C;
   // UNICODE_TO_GBK[27996] := 16#81E1;
   // UNICODE_TO_GBK[27997] := 16#C54D;
   // UNICODE_TO_GBK[27998] := 16#81E2;
   // UNICODE_TO_GBK[27999] := 16#C54E;
   // UNICODE_TO_GBK[28000] := 16#81E3;
   // UNICODE_TO_GBK[28001] := 16#B3BC;
   // UNICODE_TO_GBK[28002] := 16#81E4;
   // UNICODE_TO_GBK[28003] := 16#C54F;
   // UNICODE_TO_GBK[28004] := 16#81E5;
   // UNICODE_TO_GBK[28005] := 16#C550;
   // UNICODE_TO_GBK[28006] := 16#81E6;
   // UNICODE_TO_GBK[28007] := 16#C551;
   // UNICODE_TO_GBK[28008] := 16#81E7;
   // UNICODE_TO_GBK[28009] := 16#EAB0;
   // UNICODE_TO_GBK[28010] := 16#81E8;
   // UNICODE_TO_GBK[28011] := 16#C552;
   // UNICODE_TO_GBK[28012] := 16#81E9;
   // UNICODE_TO_GBK[28013] := 16#C553;
   // UNICODE_TO_GBK[28014] := 16#81EA;
   // UNICODE_TO_GBK[28015] := 16#D7D4;
   // UNICODE_TO_GBK[28016] := 16#81EB;
   // UNICODE_TO_GBK[28017] := 16#C554;
   // UNICODE_TO_GBK[28018] := 16#81EC;
   // UNICODE_TO_GBK[28019] := 16#F4AB;
   // UNICODE_TO_GBK[28020] := 16#81ED;
   // UNICODE_TO_GBK[28021] := 16#B3F4;
   // UNICODE_TO_GBK[28022] := 16#81EE;
   // UNICODE_TO_GBK[28023] := 16#C555;
   // UNICODE_TO_GBK[28024] := 16#81EF;
   // UNICODE_TO_GBK[28025] := 16#C556;
   // UNICODE_TO_GBK[28026] := 16#81F0;
   // UNICODE_TO_GBK[28027] := 16#C557;
   // UNICODE_TO_GBK[28028] := 16#81F1;
   // UNICODE_TO_GBK[28029] := 16#C558;
   // UNICODE_TO_GBK[28030] := 16#81F2;
   // UNICODE_TO_GBK[28031] := 16#C559;
   // UNICODE_TO_GBK[28032] := 16#81F3;
   // UNICODE_TO_GBK[28033] := 16#D6C1;
   // UNICODE_TO_GBK[28034] := 16#81F4;
   // UNICODE_TO_GBK[28035] := 16#D6C2;
   // UNICODE_TO_GBK[28036] := 16#81F5;
   // UNICODE_TO_GBK[28037] := 16#C55A;
   // UNICODE_TO_GBK[28038] := 16#81F6;
   // UNICODE_TO_GBK[28039] := 16#C55B;
   // UNICODE_TO_GBK[28040] := 16#81F7;
   // UNICODE_TO_GBK[28041] := 16#C55C;
   // UNICODE_TO_GBK[28042] := 16#81F8;
   // UNICODE_TO_GBK[28043] := 16#C55D;
   // UNICODE_TO_GBK[28044] := 16#81F9;
   // UNICODE_TO_GBK[28045] := 16#C55E;
   // UNICODE_TO_GBK[28046] := 16#81FA;
   // UNICODE_TO_GBK[28047] := 16#C55F;
   // UNICODE_TO_GBK[28048] := 16#81FB;
   // UNICODE_TO_GBK[28049] := 16#D5E9;
   // UNICODE_TO_GBK[28050] := 16#81FC;
   // UNICODE_TO_GBK[28051] := 16#BECA;
   // UNICODE_TO_GBK[28052] := 16#81FD;
   // UNICODE_TO_GBK[28053] := 16#C560;
   // UNICODE_TO_GBK[28054] := 16#81FE;
   // UNICODE_TO_GBK[28055] := 16#F4A7;
   // UNICODE_TO_GBK[28056] := 16#81FF;
   // UNICODE_TO_GBK[28057] := 16#C561;
   // UNICODE_TO_GBK[28058] := 16#8200;
   // UNICODE_TO_GBK[28059] := 16#D2A8;
   // UNICODE_TO_GBK[28060] := 16#8201;
   // UNICODE_TO_GBK[28061] := 16#F4A8;
   // UNICODE_TO_GBK[28062] := 16#8202;
   // UNICODE_TO_GBK[28063] := 16#F4A9;
   // UNICODE_TO_GBK[28064] := 16#8203;
   // UNICODE_TO_GBK[28065] := 16#C562;
   // UNICODE_TO_GBK[28066] := 16#8204;
   // UNICODE_TO_GBK[28067] := 16#F4AA;
   // UNICODE_TO_GBK[28068] := 16#8205;
   // UNICODE_TO_GBK[28069] := 16#BECB;
   // UNICODE_TO_GBK[28070] := 16#8206;
   // UNICODE_TO_GBK[28071] := 16#D3DF;
   // UNICODE_TO_GBK[28072] := 16#8207;
   // UNICODE_TO_GBK[28073] := 16#C563;
   // UNICODE_TO_GBK[28074] := 16#8208;
   // UNICODE_TO_GBK[28075] := 16#C564;
   // UNICODE_TO_GBK[28076] := 16#8209;
   // UNICODE_TO_GBK[28077] := 16#C565;
   // UNICODE_TO_GBK[28078] := 16#820A;
   // UNICODE_TO_GBK[28079] := 16#C566;
   // UNICODE_TO_GBK[28080] := 16#820B;
   // UNICODE_TO_GBK[28081] := 16#C567;
   // UNICODE_TO_GBK[28082] := 16#820C;
   // UNICODE_TO_GBK[28083] := 16#C9E0;
   // UNICODE_TO_GBK[28084] := 16#820D;
   // UNICODE_TO_GBK[28085] := 16#C9E1;
   // UNICODE_TO_GBK[28086] := 16#820E;
   // UNICODE_TO_GBK[28087] := 16#C568;
   // UNICODE_TO_GBK[28088] := 16#820F;
   // UNICODE_TO_GBK[28089] := 16#C569;
   // UNICODE_TO_GBK[28090] := 16#8210;
   // UNICODE_TO_GBK[28091] := 16#F3C2;
   // UNICODE_TO_GBK[28092] := 16#8211;
   // UNICODE_TO_GBK[28093] := 16#C56A;
   // UNICODE_TO_GBK[28094] := 16#8212;
   // UNICODE_TO_GBK[28095] := 16#CAE6;
   // UNICODE_TO_GBK[28096] := 16#8213;
   // UNICODE_TO_GBK[28097] := 16#C56B;
   // UNICODE_TO_GBK[28098] := 16#8214;
   // UNICODE_TO_GBK[28099] := 16#CCF2;
   // UNICODE_TO_GBK[28100] := 16#8215;
   // UNICODE_TO_GBK[28101] := 16#C56C;
   // UNICODE_TO_GBK[28102] := 16#8216;
   // UNICODE_TO_GBK[28103] := 16#C56D;
   // UNICODE_TO_GBK[28104] := 16#8217;
   // UNICODE_TO_GBK[28105] := 16#C56E;
   // UNICODE_TO_GBK[28106] := 16#8218;
   // UNICODE_TO_GBK[28107] := 16#C56F;
   // UNICODE_TO_GBK[28108] := 16#8219;
   // UNICODE_TO_GBK[28109] := 16#C570;
   // UNICODE_TO_GBK[28110] := 16#821A;
   // UNICODE_TO_GBK[28111] := 16#C571;
   // UNICODE_TO_GBK[28112] := 16#821B;
   // UNICODE_TO_GBK[28113] := 16#E2B6;
   // UNICODE_TO_GBK[28114] := 16#821C;
   // UNICODE_TO_GBK[28115] := 16#CBB4;
   // UNICODE_TO_GBK[28116] := 16#821D;
   // UNICODE_TO_GBK[28117] := 16#C572;
   // UNICODE_TO_GBK[28118] := 16#821E;
   // UNICODE_TO_GBK[28119] := 16#CEE8;
   // UNICODE_TO_GBK[28120] := 16#821F;
   // UNICODE_TO_GBK[28121] := 16#D6DB;
   // UNICODE_TO_GBK[28122] := 16#8220;
   // UNICODE_TO_GBK[28123] := 16#C573;
   // UNICODE_TO_GBK[28124] := 16#8221;
   // UNICODE_TO_GBK[28125] := 16#F4AD;
   // UNICODE_TO_GBK[28126] := 16#8222;
   // UNICODE_TO_GBK[28127] := 16#F4AE;
   // UNICODE_TO_GBK[28128] := 16#8223;
   // UNICODE_TO_GBK[28129] := 16#F4AF;
   // UNICODE_TO_GBK[28130] := 16#8224;
   // UNICODE_TO_GBK[28131] := 16#C574;
   // UNICODE_TO_GBK[28132] := 16#8225;
   // UNICODE_TO_GBK[28133] := 16#C575;
   // UNICODE_TO_GBK[28134] := 16#8226;
   // UNICODE_TO_GBK[28135] := 16#C576;
   // UNICODE_TO_GBK[28136] := 16#8227;
   // UNICODE_TO_GBK[28137] := 16#C577;
   // UNICODE_TO_GBK[28138] := 16#8228;
   // UNICODE_TO_GBK[28139] := 16#F4B2;
   // UNICODE_TO_GBK[28140] := 16#8229;
   // UNICODE_TO_GBK[28141] := 16#C578;
   // UNICODE_TO_GBK[28142] := 16#822A;
   // UNICODE_TO_GBK[28143] := 16#BABD;
   // UNICODE_TO_GBK[28144] := 16#822B;
   // UNICODE_TO_GBK[28145] := 16#F4B3;
   // UNICODE_TO_GBK[28146] := 16#822C;
   // UNICODE_TO_GBK[28147] := 16#B0E3;
   // UNICODE_TO_GBK[28148] := 16#822D;
   // UNICODE_TO_GBK[28149] := 16#F4B0;
   // UNICODE_TO_GBK[28150] := 16#822E;
   // UNICODE_TO_GBK[28151] := 16#C579;
   // UNICODE_TO_GBK[28152] := 16#822F;
   // UNICODE_TO_GBK[28153] := 16#F4B1;
   // UNICODE_TO_GBK[28154] := 16#8230;
   // UNICODE_TO_GBK[28155] := 16#BDA2;
   // UNICODE_TO_GBK[28156] := 16#8231;
   // UNICODE_TO_GBK[28157] := 16#B2D5;
   // UNICODE_TO_GBK[28158] := 16#8232;
   // UNICODE_TO_GBK[28159] := 16#C57A;
   // UNICODE_TO_GBK[28160] := 16#8233;
   // UNICODE_TO_GBK[28161] := 16#F4B6;
   // UNICODE_TO_GBK[28162] := 16#8234;
   // UNICODE_TO_GBK[28163] := 16#F4B7;
   // UNICODE_TO_GBK[28164] := 16#8235;
   // UNICODE_TO_GBK[28165] := 16#B6E6;
   // UNICODE_TO_GBK[28166] := 16#8236;
   // UNICODE_TO_GBK[28167] := 16#B2B0;
   // UNICODE_TO_GBK[28168] := 16#8237;
   // UNICODE_TO_GBK[28169] := 16#CFCF;
   // UNICODE_TO_GBK[28170] := 16#8238;
   // UNICODE_TO_GBK[28171] := 16#F4B4;
   // UNICODE_TO_GBK[28172] := 16#8239;
   // UNICODE_TO_GBK[28173] := 16#B4AC;
   // UNICODE_TO_GBK[28174] := 16#823A;
   // UNICODE_TO_GBK[28175] := 16#C57B;
   // UNICODE_TO_GBK[28176] := 16#823B;
   // UNICODE_TO_GBK[28177] := 16#F4B5;
   // UNICODE_TO_GBK[28178] := 16#823C;
   // UNICODE_TO_GBK[28179] := 16#C57C;
   // UNICODE_TO_GBK[28180] := 16#823D;
   // UNICODE_TO_GBK[28181] := 16#C57D;
   // UNICODE_TO_GBK[28182] := 16#823E;
   // UNICODE_TO_GBK[28183] := 16#F4B8;
   // UNICODE_TO_GBK[28184] := 16#823F;
   // UNICODE_TO_GBK[28185] := 16#C57E;
   // UNICODE_TO_GBK[28186] := 16#8240;
   // UNICODE_TO_GBK[28187] := 16#C580;
   // UNICODE_TO_GBK[28188] := 16#8241;
   // UNICODE_TO_GBK[28189] := 16#C581;
   // UNICODE_TO_GBK[28190] := 16#8242;
   // UNICODE_TO_GBK[28191] := 16#C582;
   // UNICODE_TO_GBK[28192] := 16#8243;
   // UNICODE_TO_GBK[28193] := 16#C583;
   // UNICODE_TO_GBK[28194] := 16#8244;
   // UNICODE_TO_GBK[28195] := 16#F4B9;
   // UNICODE_TO_GBK[28196] := 16#8245;
   // UNICODE_TO_GBK[28197] := 16#C584;
   // UNICODE_TO_GBK[28198] := 16#8246;
   // UNICODE_TO_GBK[28199] := 16#C585;
   // UNICODE_TO_GBK[28200] := 16#8247;
   // UNICODE_TO_GBK[28201] := 16#CDA7;
   // UNICODE_TO_GBK[28202] := 16#8248;
   // UNICODE_TO_GBK[28203] := 16#C586;
   // UNICODE_TO_GBK[28204] := 16#8249;
   // UNICODE_TO_GBK[28205] := 16#F4BA;
   // UNICODE_TO_GBK[28206] := 16#824A;
   // UNICODE_TO_GBK[28207] := 16#C587;
   // UNICODE_TO_GBK[28208] := 16#824B;
   // UNICODE_TO_GBK[28209] := 16#F4BB;
   // UNICODE_TO_GBK[28210] := 16#824C;
   // UNICODE_TO_GBK[28211] := 16#C588;
   // UNICODE_TO_GBK[28212] := 16#824D;
   // UNICODE_TO_GBK[28213] := 16#C589;
   // UNICODE_TO_GBK[28214] := 16#824E;
   // UNICODE_TO_GBK[28215] := 16#C58A;
   // UNICODE_TO_GBK[28216] := 16#824F;
   // UNICODE_TO_GBK[28217] := 16#F4BC;
   // UNICODE_TO_GBK[28218] := 16#8250;
   // UNICODE_TO_GBK[28219] := 16#C58B;
   // UNICODE_TO_GBK[28220] := 16#8251;
   // UNICODE_TO_GBK[28221] := 16#C58C;
   // UNICODE_TO_GBK[28222] := 16#8252;
   // UNICODE_TO_GBK[28223] := 16#C58D;
   // UNICODE_TO_GBK[28224] := 16#8253;
   // UNICODE_TO_GBK[28225] := 16#C58E;
   // UNICODE_TO_GBK[28226] := 16#8254;
   // UNICODE_TO_GBK[28227] := 16#C58F;
   // UNICODE_TO_GBK[28228] := 16#8255;
   // UNICODE_TO_GBK[28229] := 16#C590;
   // UNICODE_TO_GBK[28230] := 16#8256;
   // UNICODE_TO_GBK[28231] := 16#C591;
   // UNICODE_TO_GBK[28232] := 16#8257;
   // UNICODE_TO_GBK[28233] := 16#C592;
   // UNICODE_TO_GBK[28234] := 16#8258;
   // UNICODE_TO_GBK[28235] := 16#CBD2;
   // UNICODE_TO_GBK[28236] := 16#8259;
   // UNICODE_TO_GBK[28237] := 16#C593;
   // UNICODE_TO_GBK[28238] := 16#825A;
   // UNICODE_TO_GBK[28239] := 16#F4BD;
   // UNICODE_TO_GBK[28240] := 16#825B;
   // UNICODE_TO_GBK[28241] := 16#C594;
   // UNICODE_TO_GBK[28242] := 16#825C;
   // UNICODE_TO_GBK[28243] := 16#C595;
   // UNICODE_TO_GBK[28244] := 16#825D;
   // UNICODE_TO_GBK[28245] := 16#C596;
   // UNICODE_TO_GBK[28246] := 16#825E;
   // UNICODE_TO_GBK[28247] := 16#C597;
   // UNICODE_TO_GBK[28248] := 16#825F;
   // UNICODE_TO_GBK[28249] := 16#F4BE;
   // UNICODE_TO_GBK[28250] := 16#8260;
   // UNICODE_TO_GBK[28251] := 16#C598;
   // UNICODE_TO_GBK[28252] := 16#8261;
   // UNICODE_TO_GBK[28253] := 16#C599;
   // UNICODE_TO_GBK[28254] := 16#8262;
   // UNICODE_TO_GBK[28255] := 16#C59A;
   // UNICODE_TO_GBK[28256] := 16#8263;
   // UNICODE_TO_GBK[28257] := 16#C59B;
   // UNICODE_TO_GBK[28258] := 16#8264;
   // UNICODE_TO_GBK[28259] := 16#C59C;
   // UNICODE_TO_GBK[28260] := 16#8265;
   // UNICODE_TO_GBK[28261] := 16#C59D;
   // UNICODE_TO_GBK[28262] := 16#8266;
   // UNICODE_TO_GBK[28263] := 16#C59E;
   // UNICODE_TO_GBK[28264] := 16#8267;
   // UNICODE_TO_GBK[28265] := 16#C59F;
   // UNICODE_TO_GBK[28266] := 16#8268;
   // UNICODE_TO_GBK[28267] := 16#F4BF;
   // UNICODE_TO_GBK[28268] := 16#8269;
   // UNICODE_TO_GBK[28269] := 16#C5A0;
   // UNICODE_TO_GBK[28270] := 16#826A;
   // UNICODE_TO_GBK[28271] := 16#C640;
   // UNICODE_TO_GBK[28272] := 16#826B;
   // UNICODE_TO_GBK[28273] := 16#C641;
   // UNICODE_TO_GBK[28274] := 16#826C;
   // UNICODE_TO_GBK[28275] := 16#C642;
   // UNICODE_TO_GBK[28276] := 16#826D;
   // UNICODE_TO_GBK[28277] := 16#C643;
   // UNICODE_TO_GBK[28278] := 16#826E;
   // UNICODE_TO_GBK[28279] := 16#F4DE;
   // UNICODE_TO_GBK[28280] := 16#826F;
   // UNICODE_TO_GBK[28281] := 16#C1BC;
   // UNICODE_TO_GBK[28282] := 16#8270;
   // UNICODE_TO_GBK[28283] := 16#BCE8;
   // UNICODE_TO_GBK[28284] := 16#8271;
   // UNICODE_TO_GBK[28285] := 16#C644;
   // UNICODE_TO_GBK[28286] := 16#8272;
   // UNICODE_TO_GBK[28287] := 16#C9AB;
   // UNICODE_TO_GBK[28288] := 16#8273;
   // UNICODE_TO_GBK[28289] := 16#D1DE;
   // UNICODE_TO_GBK[28290] := 16#8274;
   // UNICODE_TO_GBK[28291] := 16#E5F5;
   // UNICODE_TO_GBK[28292] := 16#8275;
   // UNICODE_TO_GBK[28293] := 16#C645;
   // UNICODE_TO_GBK[28294] := 16#8276;
   // UNICODE_TO_GBK[28295] := 16#C646;
   // UNICODE_TO_GBK[28296] := 16#8277;
   // UNICODE_TO_GBK[28297] := 16#C647;
   // UNICODE_TO_GBK[28298] := 16#8278;
   // UNICODE_TO_GBK[28299] := 16#C648;
   // UNICODE_TO_GBK[28300] := 16#8279;
   // UNICODE_TO_GBK[28301] := 16#DCB3;
   // UNICODE_TO_GBK[28302] := 16#827A;
   // UNICODE_TO_GBK[28303] := 16#D2D5;
   // UNICODE_TO_GBK[28304] := 16#827B;
   // UNICODE_TO_GBK[28305] := 16#C649;
   // UNICODE_TO_GBK[28306] := 16#827C;
   // UNICODE_TO_GBK[28307] := 16#C64A;
   // UNICODE_TO_GBK[28308] := 16#827D;
   // UNICODE_TO_GBK[28309] := 16#DCB4;
   // UNICODE_TO_GBK[28310] := 16#827E;
   // UNICODE_TO_GBK[28311] := 16#B0AC;
   // UNICODE_TO_GBK[28312] := 16#827F;
   // UNICODE_TO_GBK[28313] := 16#DCB5;
   // UNICODE_TO_GBK[28314] := 16#8280;
   // UNICODE_TO_GBK[28315] := 16#C64B;
   // UNICODE_TO_GBK[28316] := 16#8281;
   // UNICODE_TO_GBK[28317] := 16#C64C;
   // UNICODE_TO_GBK[28318] := 16#8282;
   // UNICODE_TO_GBK[28319] := 16#BDDA;
   // UNICODE_TO_GBK[28320] := 16#8283;
   // UNICODE_TO_GBK[28321] := 16#C64D;
   // UNICODE_TO_GBK[28322] := 16#8284;
   // UNICODE_TO_GBK[28323] := 16#DCB9;
   // UNICODE_TO_GBK[28324] := 16#8285;
   // UNICODE_TO_GBK[28325] := 16#C64E;
   // UNICODE_TO_GBK[28326] := 16#8286;
   // UNICODE_TO_GBK[28327] := 16#C64F;
   // UNICODE_TO_GBK[28328] := 16#8287;
   // UNICODE_TO_GBK[28329] := 16#C650;
   // UNICODE_TO_GBK[28330] := 16#8288;
   // UNICODE_TO_GBK[28331] := 16#D8C2;
   // UNICODE_TO_GBK[28332] := 16#8289;
   // UNICODE_TO_GBK[28333] := 16#C651;
   // UNICODE_TO_GBK[28334] := 16#828A;
   // UNICODE_TO_GBK[28335] := 16#DCB7;
   // UNICODE_TO_GBK[28336] := 16#828B;
   // UNICODE_TO_GBK[28337] := 16#D3F3;
   // UNICODE_TO_GBK[28338] := 16#828C;
   // UNICODE_TO_GBK[28339] := 16#C652;
   // UNICODE_TO_GBK[28340] := 16#828D;
   // UNICODE_TO_GBK[28341] := 16#C9D6;
   // UNICODE_TO_GBK[28342] := 16#828E;
   // UNICODE_TO_GBK[28343] := 16#DCBA;
   // UNICODE_TO_GBK[28344] := 16#828F;
   // UNICODE_TO_GBK[28345] := 16#DCB6;
   // UNICODE_TO_GBK[28346] := 16#8290;
   // UNICODE_TO_GBK[28347] := 16#C653;
   // UNICODE_TO_GBK[28348] := 16#8291;
   // UNICODE_TO_GBK[28349] := 16#DCBB;
   // UNICODE_TO_GBK[28350] := 16#8292;
   // UNICODE_TO_GBK[28351] := 16#C3A2;
   // UNICODE_TO_GBK[28352] := 16#8293;
   // UNICODE_TO_GBK[28353] := 16#C654;
   // UNICODE_TO_GBK[28354] := 16#8294;
   // UNICODE_TO_GBK[28355] := 16#C655;
   // UNICODE_TO_GBK[28356] := 16#8295;
   // UNICODE_TO_GBK[28357] := 16#C656;
   // UNICODE_TO_GBK[28358] := 16#8296;
   // UNICODE_TO_GBK[28359] := 16#C657;
   // UNICODE_TO_GBK[28360] := 16#8297;
   // UNICODE_TO_GBK[28361] := 16#DCBC;
   // UNICODE_TO_GBK[28362] := 16#8298;
   // UNICODE_TO_GBK[28363] := 16#DCC5;
   // UNICODE_TO_GBK[28364] := 16#8299;
   // UNICODE_TO_GBK[28365] := 16#DCBD;
   // UNICODE_TO_GBK[28366] := 16#829A;
   // UNICODE_TO_GBK[28367] := 16#C658;
   // UNICODE_TO_GBK[28368] := 16#829B;
   // UNICODE_TO_GBK[28369] := 16#C659;
   // UNICODE_TO_GBK[28370] := 16#829C;
   // UNICODE_TO_GBK[28371] := 16#CEDF;
   // UNICODE_TO_GBK[28372] := 16#829D;
   // UNICODE_TO_GBK[28373] := 16#D6A5;
   // UNICODE_TO_GBK[28374] := 16#829E;
   // UNICODE_TO_GBK[28375] := 16#C65A;
   // UNICODE_TO_GBK[28376] := 16#829F;
   // UNICODE_TO_GBK[28377] := 16#DCCF;
   // UNICODE_TO_GBK[28378] := 16#82A0;
   // UNICODE_TO_GBK[28379] := 16#C65B;
   // UNICODE_TO_GBK[28380] := 16#82A1;
   // UNICODE_TO_GBK[28381] := 16#DCCD;
   // UNICODE_TO_GBK[28382] := 16#82A2;
   // UNICODE_TO_GBK[28383] := 16#C65C;
   // UNICODE_TO_GBK[28384] := 16#82A3;
   // UNICODE_TO_GBK[28385] := 16#C65D;
   // UNICODE_TO_GBK[28386] := 16#82A4;
   // UNICODE_TO_GBK[28387] := 16#DCD2;
   // UNICODE_TO_GBK[28388] := 16#82A5;
   // UNICODE_TO_GBK[28389] := 16#BDE6;
   // UNICODE_TO_GBK[28390] := 16#82A6;
   // UNICODE_TO_GBK[28391] := 16#C2AB;
   // UNICODE_TO_GBK[28392] := 16#82A7;
   // UNICODE_TO_GBK[28393] := 16#C65E;
   // UNICODE_TO_GBK[28394] := 16#82A8;
   // UNICODE_TO_GBK[28395] := 16#DCB8;
   // UNICODE_TO_GBK[28396] := 16#82A9;
   // UNICODE_TO_GBK[28397] := 16#DCCB;
   // UNICODE_TO_GBK[28398] := 16#82AA;
   // UNICODE_TO_GBK[28399] := 16#DCCE;
   // UNICODE_TO_GBK[28400] := 16#82AB;
   // UNICODE_TO_GBK[28401] := 16#DCBE;
   // UNICODE_TO_GBK[28402] := 16#82AC;
   // UNICODE_TO_GBK[28403] := 16#B7D2;
   // UNICODE_TO_GBK[28404] := 16#82AD;
   // UNICODE_TO_GBK[28405] := 16#B0C5;
   // UNICODE_TO_GBK[28406] := 16#82AE;
   // UNICODE_TO_GBK[28407] := 16#DCC7;
   // UNICODE_TO_GBK[28408] := 16#82AF;
   // UNICODE_TO_GBK[28409] := 16#D0BE;
   // UNICODE_TO_GBK[28410] := 16#82B0;
   // UNICODE_TO_GBK[28411] := 16#DCC1;
   // UNICODE_TO_GBK[28412] := 16#82B1;
   // UNICODE_TO_GBK[28413] := 16#BBA8;
   // UNICODE_TO_GBK[28414] := 16#82B2;
   // UNICODE_TO_GBK[28415] := 16#C65F;
   // UNICODE_TO_GBK[28416] := 16#82B3;
   // UNICODE_TO_GBK[28417] := 16#B7BC;
   // UNICODE_TO_GBK[28418] := 16#82B4;
   // UNICODE_TO_GBK[28419] := 16#DCCC;
   // UNICODE_TO_GBK[28420] := 16#82B5;
   // UNICODE_TO_GBK[28421] := 16#C660;
   // UNICODE_TO_GBK[28422] := 16#82B6;
   // UNICODE_TO_GBK[28423] := 16#C661;
   // UNICODE_TO_GBK[28424] := 16#82B7;
   // UNICODE_TO_GBK[28425] := 16#DCC6;
   // UNICODE_TO_GBK[28426] := 16#82B8;
   // UNICODE_TO_GBK[28427] := 16#DCBF;
   // UNICODE_TO_GBK[28428] := 16#82B9;
   // UNICODE_TO_GBK[28429] := 16#C7DB;
   // UNICODE_TO_GBK[28430] := 16#82BA;
   // UNICODE_TO_GBK[28431] := 16#C662;
   // UNICODE_TO_GBK[28432] := 16#82BB;
   // UNICODE_TO_GBK[28433] := 16#C663;
   // UNICODE_TO_GBK[28434] := 16#82BC;
   // UNICODE_TO_GBK[28435] := 16#C664;
   // UNICODE_TO_GBK[28436] := 16#82BD;
   // UNICODE_TO_GBK[28437] := 16#D1BF;
   // UNICODE_TO_GBK[28438] := 16#82BE;
   // UNICODE_TO_GBK[28439] := 16#DCC0;
   // UNICODE_TO_GBK[28440] := 16#82BF;
   // UNICODE_TO_GBK[28441] := 16#C665;
   // UNICODE_TO_GBK[28442] := 16#82C0;
   // UNICODE_TO_GBK[28443] := 16#C666;
   // UNICODE_TO_GBK[28444] := 16#82C1;
   // UNICODE_TO_GBK[28445] := 16#DCCA;
   // UNICODE_TO_GBK[28446] := 16#82C2;
   // UNICODE_TO_GBK[28447] := 16#C667;
   // UNICODE_TO_GBK[28448] := 16#82C3;
   // UNICODE_TO_GBK[28449] := 16#C668;
   // UNICODE_TO_GBK[28450] := 16#82C4;
   // UNICODE_TO_GBK[28451] := 16#DCD0;
   // UNICODE_TO_GBK[28452] := 16#82C5;
   // UNICODE_TO_GBK[28453] := 16#C669;
   // UNICODE_TO_GBK[28454] := 16#82C6;
   // UNICODE_TO_GBK[28455] := 16#C66A;
   // UNICODE_TO_GBK[28456] := 16#82C7;
   // UNICODE_TO_GBK[28457] := 16#CEAD;
   // UNICODE_TO_GBK[28458] := 16#82C8;
   // UNICODE_TO_GBK[28459] := 16#DCC2;
   // UNICODE_TO_GBK[28460] := 16#82C9;
   // UNICODE_TO_GBK[28461] := 16#C66B;
   // UNICODE_TO_GBK[28462] := 16#82CA;
   // UNICODE_TO_GBK[28463] := 16#DCC3;
   // UNICODE_TO_GBK[28464] := 16#82CB;
   // UNICODE_TO_GBK[28465] := 16#DCC8;
   // UNICODE_TO_GBK[28466] := 16#82CC;
   // UNICODE_TO_GBK[28467] := 16#DCC9;
   // UNICODE_TO_GBK[28468] := 16#82CD;
   // UNICODE_TO_GBK[28469] := 16#B2D4;
   // UNICODE_TO_GBK[28470] := 16#82CE;
   // UNICODE_TO_GBK[28471] := 16#DCD1;
   // UNICODE_TO_GBK[28472] := 16#82CF;
   // UNICODE_TO_GBK[28473] := 16#CBD5;
   // UNICODE_TO_GBK[28474] := 16#82D0;
   // UNICODE_TO_GBK[28475] := 16#C66C;
   // UNICODE_TO_GBK[28476] := 16#82D1;
   // UNICODE_TO_GBK[28477] := 16#D4B7;
   // UNICODE_TO_GBK[28478] := 16#82D2;
   // UNICODE_TO_GBK[28479] := 16#DCDB;
   // UNICODE_TO_GBK[28480] := 16#82D3;
   // UNICODE_TO_GBK[28481] := 16#DCDF;
   // UNICODE_TO_GBK[28482] := 16#82D4;
   // UNICODE_TO_GBK[28483] := 16#CCA6;
   // UNICODE_TO_GBK[28484] := 16#82D5;
   // UNICODE_TO_GBK[28485] := 16#DCE6;
   // UNICODE_TO_GBK[28486] := 16#82D6;
   // UNICODE_TO_GBK[28487] := 16#C66D;
   // UNICODE_TO_GBK[28488] := 16#82D7;
   // UNICODE_TO_GBK[28489] := 16#C3E7;
   // UNICODE_TO_GBK[28490] := 16#82D8;
   // UNICODE_TO_GBK[28491] := 16#DCDC;
   // UNICODE_TO_GBK[28492] := 16#82D9;
   // UNICODE_TO_GBK[28493] := 16#C66E;
   // UNICODE_TO_GBK[28494] := 16#82DA;
   // UNICODE_TO_GBK[28495] := 16#C66F;
   // UNICODE_TO_GBK[28496] := 16#82DB;
   // UNICODE_TO_GBK[28497] := 16#BFC1;
   // UNICODE_TO_GBK[28498] := 16#82DC;
   // UNICODE_TO_GBK[28499] := 16#DCD9;
   // UNICODE_TO_GBK[28500] := 16#82DD;
   // UNICODE_TO_GBK[28501] := 16#C670;
   // UNICODE_TO_GBK[28502] := 16#82DE;
   // UNICODE_TO_GBK[28503] := 16#B0FA;
   // UNICODE_TO_GBK[28504] := 16#82DF;
   // UNICODE_TO_GBK[28505] := 16#B9B6;
   // UNICODE_TO_GBK[28506] := 16#82E0;
   // UNICODE_TO_GBK[28507] := 16#DCE5;
   // UNICODE_TO_GBK[28508] := 16#82E1;
   // UNICODE_TO_GBK[28509] := 16#DCD3;
   // UNICODE_TO_GBK[28510] := 16#82E2;
   // UNICODE_TO_GBK[28511] := 16#C671;
   // UNICODE_TO_GBK[28512] := 16#82E3;
   // UNICODE_TO_GBK[28513] := 16#DCC4;
   // UNICODE_TO_GBK[28514] := 16#82E4;
   // UNICODE_TO_GBK[28515] := 16#DCD6;
   // UNICODE_TO_GBK[28516] := 16#82E5;
   // UNICODE_TO_GBK[28517] := 16#C8F4;
   // UNICODE_TO_GBK[28518] := 16#82E6;
   // UNICODE_TO_GBK[28519] := 16#BFE0;
   // UNICODE_TO_GBK[28520] := 16#82E7;
   // UNICODE_TO_GBK[28521] := 16#C672;
   // UNICODE_TO_GBK[28522] := 16#82E8;
   // UNICODE_TO_GBK[28523] := 16#C673;
   // UNICODE_TO_GBK[28524] := 16#82E9;
   // UNICODE_TO_GBK[28525] := 16#C674;
   // UNICODE_TO_GBK[28526] := 16#82EA;
   // UNICODE_TO_GBK[28527] := 16#C675;
   // UNICODE_TO_GBK[28528] := 16#82EB;
   // UNICODE_TO_GBK[28529] := 16#C9BB;
   // UNICODE_TO_GBK[28530] := 16#82EC;
   // UNICODE_TO_GBK[28531] := 16#C676;
   // UNICODE_TO_GBK[28532] := 16#82ED;
   // UNICODE_TO_GBK[28533] := 16#C677;
   // UNICODE_TO_GBK[28534] := 16#82EE;
   // UNICODE_TO_GBK[28535] := 16#C678;
   // UNICODE_TO_GBK[28536] := 16#82EF;
   // UNICODE_TO_GBK[28537] := 16#B1BD;
   // UNICODE_TO_GBK[28538] := 16#82F0;
   // UNICODE_TO_GBK[28539] := 16#C679;
   // UNICODE_TO_GBK[28540] := 16#82F1;
   // UNICODE_TO_GBK[28541] := 16#D3A2;
   // UNICODE_TO_GBK[28542] := 16#82F2;
   // UNICODE_TO_GBK[28543] := 16#C67A;
   // UNICODE_TO_GBK[28544] := 16#82F3;
   // UNICODE_TO_GBK[28545] := 16#C67B;
   // UNICODE_TO_GBK[28546] := 16#82F4;
   // UNICODE_TO_GBK[28547] := 16#DCDA;
   // UNICODE_TO_GBK[28548] := 16#82F5;
   // UNICODE_TO_GBK[28549] := 16#C67C;
   // UNICODE_TO_GBK[28550] := 16#82F6;
   // UNICODE_TO_GBK[28551] := 16#C67D;
   // UNICODE_TO_GBK[28552] := 16#82F7;
   // UNICODE_TO_GBK[28553] := 16#DCD5;
   // UNICODE_TO_GBK[28554] := 16#82F8;
   // UNICODE_TO_GBK[28555] := 16#C67E;
   // UNICODE_TO_GBK[28556] := 16#82F9;
   // UNICODE_TO_GBK[28557] := 16#C6BB;
   // UNICODE_TO_GBK[28558] := 16#82FA;
   // UNICODE_TO_GBK[28559] := 16#C680;
   // UNICODE_TO_GBK[28560] := 16#82FB;
   // UNICODE_TO_GBK[28561] := 16#DCDE;
   // UNICODE_TO_GBK[28562] := 16#82FC;
   // UNICODE_TO_GBK[28563] := 16#C681;
   // UNICODE_TO_GBK[28564] := 16#82FD;
   // UNICODE_TO_GBK[28565] := 16#C682;
   // UNICODE_TO_GBK[28566] := 16#82FE;
   // UNICODE_TO_GBK[28567] := 16#C683;
   // UNICODE_TO_GBK[28568] := 16#82FF;
   // UNICODE_TO_GBK[28569] := 16#C684;
   // UNICODE_TO_GBK[28570] := 16#8300;
   // UNICODE_TO_GBK[28571] := 16#C685;
   // UNICODE_TO_GBK[28572] := 16#8301;
   // UNICODE_TO_GBK[28573] := 16#D7C2;
   // UNICODE_TO_GBK[28574] := 16#8302;
   // UNICODE_TO_GBK[28575] := 16#C3AF;
   // UNICODE_TO_GBK[28576] := 16#8303;
   // UNICODE_TO_GBK[28577] := 16#B7B6;
   // UNICODE_TO_GBK[28578] := 16#8304;
   // UNICODE_TO_GBK[28579] := 16#C7D1;
   // UNICODE_TO_GBK[28580] := 16#8305;
   // UNICODE_TO_GBK[28581] := 16#C3A9;
   // UNICODE_TO_GBK[28582] := 16#8306;
   // UNICODE_TO_GBK[28583] := 16#DCE2;
   // UNICODE_TO_GBK[28584] := 16#8307;
   // UNICODE_TO_GBK[28585] := 16#DCD8;
   // UNICODE_TO_GBK[28586] := 16#8308;
   // UNICODE_TO_GBK[28587] := 16#DCEB;
   // UNICODE_TO_GBK[28588] := 16#8309;
   // UNICODE_TO_GBK[28589] := 16#DCD4;
   // UNICODE_TO_GBK[28590] := 16#830A;
   // UNICODE_TO_GBK[28591] := 16#C686;
   // UNICODE_TO_GBK[28592] := 16#830B;
   // UNICODE_TO_GBK[28593] := 16#C687;
   // UNICODE_TO_GBK[28594] := 16#830C;
   // UNICODE_TO_GBK[28595] := 16#DCDD;
   // UNICODE_TO_GBK[28596] := 16#830D;
   // UNICODE_TO_GBK[28597] := 16#C688;
   // UNICODE_TO_GBK[28598] := 16#830E;
   // UNICODE_TO_GBK[28599] := 16#BEA5;
   // UNICODE_TO_GBK[28600] := 16#830F;
   // UNICODE_TO_GBK[28601] := 16#DCD7;
   // UNICODE_TO_GBK[28602] := 16#8310;
   // UNICODE_TO_GBK[28603] := 16#C689;
   // UNICODE_TO_GBK[28604] := 16#8311;
   // UNICODE_TO_GBK[28605] := 16#DCE0;
   // UNICODE_TO_GBK[28606] := 16#8312;
   // UNICODE_TO_GBK[28607] := 16#C68A;
   // UNICODE_TO_GBK[28608] := 16#8313;
   // UNICODE_TO_GBK[28609] := 16#C68B;
   // UNICODE_TO_GBK[28610] := 16#8314;
   // UNICODE_TO_GBK[28611] := 16#DCE3;
   // UNICODE_TO_GBK[28612] := 16#8315;
   // UNICODE_TO_GBK[28613] := 16#DCE4;
   // UNICODE_TO_GBK[28614] := 16#8316;
   // UNICODE_TO_GBK[28615] := 16#C68C;
   // UNICODE_TO_GBK[28616] := 16#8317;
   // UNICODE_TO_GBK[28617] := 16#DCF8;
   // UNICODE_TO_GBK[28618] := 16#8318;
   // UNICODE_TO_GBK[28619] := 16#C68D;
   // UNICODE_TO_GBK[28620] := 16#8319;
   // UNICODE_TO_GBK[28621] := 16#C68E;
   // UNICODE_TO_GBK[28622] := 16#831A;
   // UNICODE_TO_GBK[28623] := 16#DCE1;
   // UNICODE_TO_GBK[28624] := 16#831B;
   // UNICODE_TO_GBK[28625] := 16#DDA2;
   // UNICODE_TO_GBK[28626] := 16#831C;
   // UNICODE_TO_GBK[28627] := 16#DCE7;
   // UNICODE_TO_GBK[28628] := 16#831D;
   // UNICODE_TO_GBK[28629] := 16#C68F;
   // UNICODE_TO_GBK[28630] := 16#831E;
   // UNICODE_TO_GBK[28631] := 16#C690;
   // UNICODE_TO_GBK[28632] := 16#831F;
   // UNICODE_TO_GBK[28633] := 16#C691;
   // UNICODE_TO_GBK[28634] := 16#8320;
   // UNICODE_TO_GBK[28635] := 16#C692;
   // UNICODE_TO_GBK[28636] := 16#8321;
   // UNICODE_TO_GBK[28637] := 16#C693;
   // UNICODE_TO_GBK[28638] := 16#8322;
   // UNICODE_TO_GBK[28639] := 16#C694;
   // UNICODE_TO_GBK[28640] := 16#8323;
   // UNICODE_TO_GBK[28641] := 16#C695;
   // UNICODE_TO_GBK[28642] := 16#8324;
   // UNICODE_TO_GBK[28643] := 16#C696;
   // UNICODE_TO_GBK[28644] := 16#8325;
   // UNICODE_TO_GBK[28645] := 16#C697;
   // UNICODE_TO_GBK[28646] := 16#8326;
   // UNICODE_TO_GBK[28647] := 16#C698;
   // UNICODE_TO_GBK[28648] := 16#8327;
   // UNICODE_TO_GBK[28649] := 16#BCEB;
   // UNICODE_TO_GBK[28650] := 16#8328;
   // UNICODE_TO_GBK[28651] := 16#B4C4;
   // UNICODE_TO_GBK[28652] := 16#8329;
   // UNICODE_TO_GBK[28653] := 16#C699;
   // UNICODE_TO_GBK[28654] := 16#832A;
   // UNICODE_TO_GBK[28655] := 16#C69A;
   // UNICODE_TO_GBK[28656] := 16#832B;
   // UNICODE_TO_GBK[28657] := 16#C3A3;
   // UNICODE_TO_GBK[28658] := 16#832C;
   // UNICODE_TO_GBK[28659] := 16#B2E7;
   // UNICODE_TO_GBK[28660] := 16#832D;
   // UNICODE_TO_GBK[28661] := 16#DCFA;
   // UNICODE_TO_GBK[28662] := 16#832E;
   // UNICODE_TO_GBK[28663] := 16#C69B;
   // UNICODE_TO_GBK[28664] := 16#832F;
   // UNICODE_TO_GBK[28665] := 16#DCF2;
   // UNICODE_TO_GBK[28666] := 16#8330;
   // UNICODE_TO_GBK[28667] := 16#C69C;
   // UNICODE_TO_GBK[28668] := 16#8331;
   // UNICODE_TO_GBK[28669] := 16#DCEF;
   // UNICODE_TO_GBK[28670] := 16#8332;
   // UNICODE_TO_GBK[28671] := 16#C69D;
   // UNICODE_TO_GBK[28672] := 16#8333;
   // UNICODE_TO_GBK[28673] := 16#DCFC;
   // UNICODE_TO_GBK[28674] := 16#8334;
   // UNICODE_TO_GBK[28675] := 16#DCEE;
   // UNICODE_TO_GBK[28676] := 16#8335;
   // UNICODE_TO_GBK[28677] := 16#D2F0;
   // UNICODE_TO_GBK[28678] := 16#8336;
   // UNICODE_TO_GBK[28679] := 16#B2E8;
   // UNICODE_TO_GBK[28680] := 16#8337;
   // UNICODE_TO_GBK[28681] := 16#C69E;
   // UNICODE_TO_GBK[28682] := 16#8338;
   // UNICODE_TO_GBK[28683] := 16#C8D7;
   // UNICODE_TO_GBK[28684] := 16#8339;
   // UNICODE_TO_GBK[28685] := 16#C8E3;
   // UNICODE_TO_GBK[28686] := 16#833A;
   // UNICODE_TO_GBK[28687] := 16#DCFB;
   // UNICODE_TO_GBK[28688] := 16#833B;
   // UNICODE_TO_GBK[28689] := 16#C69F;
   // UNICODE_TO_GBK[28690] := 16#833C;
   // UNICODE_TO_GBK[28691] := 16#DCED;
   // UNICODE_TO_GBK[28692] := 16#833D;
   // UNICODE_TO_GBK[28693] := 16#C6A0;
   // UNICODE_TO_GBK[28694] := 16#833E;
   // UNICODE_TO_GBK[28695] := 16#C740;
   // UNICODE_TO_GBK[28696] := 16#833F;
   // UNICODE_TO_GBK[28697] := 16#C741;
   // UNICODE_TO_GBK[28698] := 16#8340;
   // UNICODE_TO_GBK[28699] := 16#DCF7;
   // UNICODE_TO_GBK[28700] := 16#8341;
   // UNICODE_TO_GBK[28701] := 16#C742;
   // UNICODE_TO_GBK[28702] := 16#8342;
   // UNICODE_TO_GBK[28703] := 16#C743;
   // UNICODE_TO_GBK[28704] := 16#8343;
   // UNICODE_TO_GBK[28705] := 16#DCF5;
   // UNICODE_TO_GBK[28706] := 16#8344;
   // UNICODE_TO_GBK[28707] := 16#C744;
   // UNICODE_TO_GBK[28708] := 16#8345;
   // UNICODE_TO_GBK[28709] := 16#C745;
   // UNICODE_TO_GBK[28710] := 16#8346;
   // UNICODE_TO_GBK[28711] := 16#BEA3;
   // UNICODE_TO_GBK[28712] := 16#8347;
   // UNICODE_TO_GBK[28713] := 16#DCF4;
   // UNICODE_TO_GBK[28714] := 16#8348;
   // UNICODE_TO_GBK[28715] := 16#C746;
   // UNICODE_TO_GBK[28716] := 16#8349;
   // UNICODE_TO_GBK[28717] := 16#B2DD;
   // UNICODE_TO_GBK[28718] := 16#834A;
   // UNICODE_TO_GBK[28719] := 16#C747;
   // UNICODE_TO_GBK[28720] := 16#834B;
   // UNICODE_TO_GBK[28721] := 16#C748;
   // UNICODE_TO_GBK[28722] := 16#834C;
   // UNICODE_TO_GBK[28723] := 16#C749;
   // UNICODE_TO_GBK[28724] := 16#834D;
   // UNICODE_TO_GBK[28725] := 16#C74A;
   // UNICODE_TO_GBK[28726] := 16#834E;
   // UNICODE_TO_GBK[28727] := 16#C74B;
   // UNICODE_TO_GBK[28728] := 16#834F;
   // UNICODE_TO_GBK[28729] := 16#DCF3;
   // UNICODE_TO_GBK[28730] := 16#8350;
   // UNICODE_TO_GBK[28731] := 16#BCF6;
   // UNICODE_TO_GBK[28732] := 16#8351;
   // UNICODE_TO_GBK[28733] := 16#DCE8;
   // UNICODE_TO_GBK[28734] := 16#8352;
   // UNICODE_TO_GBK[28735] := 16#BBC4;
   // UNICODE_TO_GBK[28736] := 16#8353;
   // UNICODE_TO_GBK[28737] := 16#C74C;
   // UNICODE_TO_GBK[28738] := 16#8354;
   // UNICODE_TO_GBK[28739] := 16#C0F3;
   // UNICODE_TO_GBK[28740] := 16#8355;
   // UNICODE_TO_GBK[28741] := 16#C74D;
   // UNICODE_TO_GBK[28742] := 16#8356;
   // UNICODE_TO_GBK[28743] := 16#C74E;
   // UNICODE_TO_GBK[28744] := 16#8357;
   // UNICODE_TO_GBK[28745] := 16#C74F;
   // UNICODE_TO_GBK[28746] := 16#8358;
   // UNICODE_TO_GBK[28747] := 16#C750;
   // UNICODE_TO_GBK[28748] := 16#8359;
   // UNICODE_TO_GBK[28749] := 16#C751;
   // UNICODE_TO_GBK[28750] := 16#835A;
   // UNICODE_TO_GBK[28751] := 16#BCD4;
   // UNICODE_TO_GBK[28752] := 16#835B;
   // UNICODE_TO_GBK[28753] := 16#DCE9;
   // UNICODE_TO_GBK[28754] := 16#835C;
   // UNICODE_TO_GBK[28755] := 16#DCEA;
   // UNICODE_TO_GBK[28756] := 16#835D;
   // UNICODE_TO_GBK[28757] := 16#C752;
   // UNICODE_TO_GBK[28758] := 16#835E;
   // UNICODE_TO_GBK[28759] := 16#DCF1;
   // UNICODE_TO_GBK[28760] := 16#835F;
   // UNICODE_TO_GBK[28761] := 16#DCF6;
   // UNICODE_TO_GBK[28762] := 16#8360;
   // UNICODE_TO_GBK[28763] := 16#DCF9;
   // UNICODE_TO_GBK[28764] := 16#8361;
   // UNICODE_TO_GBK[28765] := 16#B5B4;
   // UNICODE_TO_GBK[28766] := 16#8362;
   // UNICODE_TO_GBK[28767] := 16#C753;
   // UNICODE_TO_GBK[28768] := 16#8363;
   // UNICODE_TO_GBK[28769] := 16#C8D9;
   // UNICODE_TO_GBK[28770] := 16#8364;
   // UNICODE_TO_GBK[28771] := 16#BBE7;
   // UNICODE_TO_GBK[28772] := 16#8365;
   // UNICODE_TO_GBK[28773] := 16#DCFE;
   // UNICODE_TO_GBK[28774] := 16#8366;
   // UNICODE_TO_GBK[28775] := 16#DCFD;
   // UNICODE_TO_GBK[28776] := 16#8367;
   // UNICODE_TO_GBK[28777] := 16#D3AB;
   // UNICODE_TO_GBK[28778] := 16#8368;
   // UNICODE_TO_GBK[28779] := 16#DDA1;
   // UNICODE_TO_GBK[28780] := 16#8369;
   // UNICODE_TO_GBK[28781] := 16#DDA3;
   // UNICODE_TO_GBK[28782] := 16#836A;
   // UNICODE_TO_GBK[28783] := 16#DDA5;
   // UNICODE_TO_GBK[28784] := 16#836B;
   // UNICODE_TO_GBK[28785] := 16#D2F1;
   // UNICODE_TO_GBK[28786] := 16#836C;
   // UNICODE_TO_GBK[28787] := 16#DDA4;
   // UNICODE_TO_GBK[28788] := 16#836D;
   // UNICODE_TO_GBK[28789] := 16#DDA6;
   // UNICODE_TO_GBK[28790] := 16#836E;
   // UNICODE_TO_GBK[28791] := 16#DDA7;
   // UNICODE_TO_GBK[28792] := 16#836F;
   // UNICODE_TO_GBK[28793] := 16#D2A9;
   // UNICODE_TO_GBK[28794] := 16#8370;
   // UNICODE_TO_GBK[28795] := 16#C754;
   // UNICODE_TO_GBK[28796] := 16#8371;
   // UNICODE_TO_GBK[28797] := 16#C755;
   // UNICODE_TO_GBK[28798] := 16#8372;
   // UNICODE_TO_GBK[28799] := 16#C756;
   // UNICODE_TO_GBK[28800] := 16#8373;
   // UNICODE_TO_GBK[28801] := 16#C757;
   // UNICODE_TO_GBK[28802] := 16#8374;
   // UNICODE_TO_GBK[28803] := 16#C758;
   // UNICODE_TO_GBK[28804] := 16#8375;
   // UNICODE_TO_GBK[28805] := 16#C759;
   // UNICODE_TO_GBK[28806] := 16#8376;
   // UNICODE_TO_GBK[28807] := 16#C75A;
   // UNICODE_TO_GBK[28808] := 16#8377;
   // UNICODE_TO_GBK[28809] := 16#BAC9;
   // UNICODE_TO_GBK[28810] := 16#8378;
   // UNICODE_TO_GBK[28811] := 16#DDA9;
   // UNICODE_TO_GBK[28812] := 16#8379;
   // UNICODE_TO_GBK[28813] := 16#C75B;
   // UNICODE_TO_GBK[28814] := 16#837A;
   // UNICODE_TO_GBK[28815] := 16#C75C;
   // UNICODE_TO_GBK[28816] := 16#837B;
   // UNICODE_TO_GBK[28817] := 16#DDB6;
   // UNICODE_TO_GBK[28818] := 16#837C;
   // UNICODE_TO_GBK[28819] := 16#DDB1;
   // UNICODE_TO_GBK[28820] := 16#837D;
   // UNICODE_TO_GBK[28821] := 16#DDB4;
   // UNICODE_TO_GBK[28822] := 16#837E;
   // UNICODE_TO_GBK[28823] := 16#C75D;
   // UNICODE_TO_GBK[28824] := 16#837F;
   // UNICODE_TO_GBK[28825] := 16#C75E;
   // UNICODE_TO_GBK[28826] := 16#8380;
   // UNICODE_TO_GBK[28827] := 16#C75F;
   // UNICODE_TO_GBK[28828] := 16#8381;
   // UNICODE_TO_GBK[28829] := 16#C760;
   // UNICODE_TO_GBK[28830] := 16#8382;
   // UNICODE_TO_GBK[28831] := 16#C761;
   // UNICODE_TO_GBK[28832] := 16#8383;
   // UNICODE_TO_GBK[28833] := 16#C762;
   // UNICODE_TO_GBK[28834] := 16#8384;
   // UNICODE_TO_GBK[28835] := 16#C763;
   // UNICODE_TO_GBK[28836] := 16#8385;
   // UNICODE_TO_GBK[28837] := 16#DDB0;
   // UNICODE_TO_GBK[28838] := 16#8386;
   // UNICODE_TO_GBK[28839] := 16#C6CE;
   // UNICODE_TO_GBK[28840] := 16#8387;
   // UNICODE_TO_GBK[28841] := 16#C764;
   // UNICODE_TO_GBK[28842] := 16#8388;
   // UNICODE_TO_GBK[28843] := 16#C765;
   // UNICODE_TO_GBK[28844] := 16#8389;
   // UNICODE_TO_GBK[28845] := 16#C0F2;
   // UNICODE_TO_GBK[28846] := 16#838A;
   // UNICODE_TO_GBK[28847] := 16#C766;
   // UNICODE_TO_GBK[28848] := 16#838B;
   // UNICODE_TO_GBK[28849] := 16#C767;
   // UNICODE_TO_GBK[28850] := 16#838C;
   // UNICODE_TO_GBK[28851] := 16#C768;
   // UNICODE_TO_GBK[28852] := 16#838D;
   // UNICODE_TO_GBK[28853] := 16#C769;
   // UNICODE_TO_GBK[28854] := 16#838E;
   // UNICODE_TO_GBK[28855] := 16#C9AF;
   // UNICODE_TO_GBK[28856] := 16#838F;
   // UNICODE_TO_GBK[28857] := 16#C76A;
   // UNICODE_TO_GBK[28858] := 16#8390;
   // UNICODE_TO_GBK[28859] := 16#C76B;
   // UNICODE_TO_GBK[28860] := 16#8391;
   // UNICODE_TO_GBK[28861] := 16#C76C;
   // UNICODE_TO_GBK[28862] := 16#8392;
   // UNICODE_TO_GBK[28863] := 16#DCEC;
   // UNICODE_TO_GBK[28864] := 16#8393;
   // UNICODE_TO_GBK[28865] := 16#DDAE;
   // UNICODE_TO_GBK[28866] := 16#8394;
   // UNICODE_TO_GBK[28867] := 16#C76D;
   // UNICODE_TO_GBK[28868] := 16#8395;
   // UNICODE_TO_GBK[28869] := 16#C76E;
   // UNICODE_TO_GBK[28870] := 16#8396;
   // UNICODE_TO_GBK[28871] := 16#C76F;
   // UNICODE_TO_GBK[28872] := 16#8397;
   // UNICODE_TO_GBK[28873] := 16#C770;
   // UNICODE_TO_GBK[28874] := 16#8398;
   // UNICODE_TO_GBK[28875] := 16#DDB7;
   // UNICODE_TO_GBK[28876] := 16#8399;
   // UNICODE_TO_GBK[28877] := 16#C771;
   // UNICODE_TO_GBK[28878] := 16#839A;
   // UNICODE_TO_GBK[28879] := 16#C772;
   // UNICODE_TO_GBK[28880] := 16#839B;
   // UNICODE_TO_GBK[28881] := 16#DCF0;
   // UNICODE_TO_GBK[28882] := 16#839C;
   // UNICODE_TO_GBK[28883] := 16#DDAF;
   // UNICODE_TO_GBK[28884] := 16#839D;
   // UNICODE_TO_GBK[28885] := 16#C773;
   // UNICODE_TO_GBK[28886] := 16#839E;
   // UNICODE_TO_GBK[28887] := 16#DDB8;
   // UNICODE_TO_GBK[28888] := 16#839F;
   // UNICODE_TO_GBK[28889] := 16#C774;
   // UNICODE_TO_GBK[28890] := 16#83A0;
   // UNICODE_TO_GBK[28891] := 16#DDAC;
   // UNICODE_TO_GBK[28892] := 16#83A1;
   // UNICODE_TO_GBK[28893] := 16#C775;
   // UNICODE_TO_GBK[28894] := 16#83A2;
   // UNICODE_TO_GBK[28895] := 16#C776;
   // UNICODE_TO_GBK[28896] := 16#83A3;
   // UNICODE_TO_GBK[28897] := 16#C777;
   // UNICODE_TO_GBK[28898] := 16#83A4;
   // UNICODE_TO_GBK[28899] := 16#C778;
   // UNICODE_TO_GBK[28900] := 16#83A5;
   // UNICODE_TO_GBK[28901] := 16#C779;
   // UNICODE_TO_GBK[28902] := 16#83A6;
   // UNICODE_TO_GBK[28903] := 16#C77A;
   // UNICODE_TO_GBK[28904] := 16#83A7;
   // UNICODE_TO_GBK[28905] := 16#C77B;
   // UNICODE_TO_GBK[28906] := 16#83A8;
   // UNICODE_TO_GBK[28907] := 16#DDB9;
   // UNICODE_TO_GBK[28908] := 16#83A9;
   // UNICODE_TO_GBK[28909] := 16#DDB3;
   // UNICODE_TO_GBK[28910] := 16#83AA;
   // UNICODE_TO_GBK[28911] := 16#DDAD;
   // UNICODE_TO_GBK[28912] := 16#83AB;
   // UNICODE_TO_GBK[28913] := 16#C4AA;
   // UNICODE_TO_GBK[28914] := 16#83AC;
   // UNICODE_TO_GBK[28915] := 16#C77C;
   // UNICODE_TO_GBK[28916] := 16#83AD;
   // UNICODE_TO_GBK[28917] := 16#C77D;
   // UNICODE_TO_GBK[28918] := 16#83AE;
   // UNICODE_TO_GBK[28919] := 16#C77E;
   // UNICODE_TO_GBK[28920] := 16#83AF;
   // UNICODE_TO_GBK[28921] := 16#C780;
   // UNICODE_TO_GBK[28922] := 16#83B0;
   // UNICODE_TO_GBK[28923] := 16#DDA8;
   // UNICODE_TO_GBK[28924] := 16#83B1;
   // UNICODE_TO_GBK[28925] := 16#C0B3;
   // UNICODE_TO_GBK[28926] := 16#83B2;
   // UNICODE_TO_GBK[28927] := 16#C1AB;
   // UNICODE_TO_GBK[28928] := 16#83B3;
   // UNICODE_TO_GBK[28929] := 16#DDAA;
   // UNICODE_TO_GBK[28930] := 16#83B4;
   // UNICODE_TO_GBK[28931] := 16#DDAB;
   // UNICODE_TO_GBK[28932] := 16#83B5;
   // UNICODE_TO_GBK[28933] := 16#C781;
   // UNICODE_TO_GBK[28934] := 16#83B6;
   // UNICODE_TO_GBK[28935] := 16#DDB2;
   // UNICODE_TO_GBK[28936] := 16#83B7;
   // UNICODE_TO_GBK[28937] := 16#BBF1;
   // UNICODE_TO_GBK[28938] := 16#83B8;
   // UNICODE_TO_GBK[28939] := 16#DDB5;
   // UNICODE_TO_GBK[28940] := 16#83B9;
   // UNICODE_TO_GBK[28941] := 16#D3A8;
   // UNICODE_TO_GBK[28942] := 16#83BA;
   // UNICODE_TO_GBK[28943] := 16#DDBA;
   // UNICODE_TO_GBK[28944] := 16#83BB;
   // UNICODE_TO_GBK[28945] := 16#C782;
   // UNICODE_TO_GBK[28946] := 16#83BC;
   // UNICODE_TO_GBK[28947] := 16#DDBB;
   // UNICODE_TO_GBK[28948] := 16#83BD;
   // UNICODE_TO_GBK[28949] := 16#C3A7;
   // UNICODE_TO_GBK[28950] := 16#83BE;
   // UNICODE_TO_GBK[28951] := 16#C783;
   // UNICODE_TO_GBK[28952] := 16#83BF;
   // UNICODE_TO_GBK[28953] := 16#C784;
   // UNICODE_TO_GBK[28954] := 16#83C0;
   // UNICODE_TO_GBK[28955] := 16#DDD2;
   // UNICODE_TO_GBK[28956] := 16#83C1;
   // UNICODE_TO_GBK[28957] := 16#DDBC;
   // UNICODE_TO_GBK[28958] := 16#83C2;
   // UNICODE_TO_GBK[28959] := 16#C785;
   // UNICODE_TO_GBK[28960] := 16#83C3;
   // UNICODE_TO_GBK[28961] := 16#C786;
   // UNICODE_TO_GBK[28962] := 16#83C4;
   // UNICODE_TO_GBK[28963] := 16#C787;
   // UNICODE_TO_GBK[28964] := 16#83C5;
   // UNICODE_TO_GBK[28965] := 16#DDD1;
   // UNICODE_TO_GBK[28966] := 16#83C6;
   // UNICODE_TO_GBK[28967] := 16#C788;
   // UNICODE_TO_GBK[28968] := 16#83C7;
   // UNICODE_TO_GBK[28969] := 16#B9BD;
   // UNICODE_TO_GBK[28970] := 16#83C8;
   // UNICODE_TO_GBK[28971] := 16#C789;
   // UNICODE_TO_GBK[28972] := 16#83C9;
   // UNICODE_TO_GBK[28973] := 16#C78A;
   // UNICODE_TO_GBK[28974] := 16#83CA;
   // UNICODE_TO_GBK[28975] := 16#BED5;
   // UNICODE_TO_GBK[28976] := 16#83CB;
   // UNICODE_TO_GBK[28977] := 16#C78B;
   // UNICODE_TO_GBK[28978] := 16#83CC;
   // UNICODE_TO_GBK[28979] := 16#BEFA;
   // UNICODE_TO_GBK[28980] := 16#83CD;
   // UNICODE_TO_GBK[28981] := 16#C78C;
   // UNICODE_TO_GBK[28982] := 16#83CE;
   // UNICODE_TO_GBK[28983] := 16#C78D;
   // UNICODE_TO_GBK[28984] := 16#83CF;
   // UNICODE_TO_GBK[28985] := 16#BACA;
   // UNICODE_TO_GBK[28986] := 16#83D0;
   // UNICODE_TO_GBK[28987] := 16#C78E;
   // UNICODE_TO_GBK[28988] := 16#83D1;
   // UNICODE_TO_GBK[28989] := 16#C78F;
   // UNICODE_TO_GBK[28990] := 16#83D2;
   // UNICODE_TO_GBK[28991] := 16#C790;
   // UNICODE_TO_GBK[28992] := 16#83D3;
   // UNICODE_TO_GBK[28993] := 16#C791;
   // UNICODE_TO_GBK[28994] := 16#83D4;
   // UNICODE_TO_GBK[28995] := 16#DDCA;
   // UNICODE_TO_GBK[28996] := 16#83D5;
   // UNICODE_TO_GBK[28997] := 16#C792;
   // UNICODE_TO_GBK[28998] := 16#83D6;
   // UNICODE_TO_GBK[28999] := 16#DDC5;
   // UNICODE_TO_GBK[29000] := 16#83D7;
   // UNICODE_TO_GBK[29001] := 16#C793;
   // UNICODE_TO_GBK[29002] := 16#83D8;
   // UNICODE_TO_GBK[29003] := 16#DDBF;
   // UNICODE_TO_GBK[29004] := 16#83D9;
   // UNICODE_TO_GBK[29005] := 16#C794;
   // UNICODE_TO_GBK[29006] := 16#83DA;
   // UNICODE_TO_GBK[29007] := 16#C795;
   // UNICODE_TO_GBK[29008] := 16#83DB;
   // UNICODE_TO_GBK[29009] := 16#C796;
   // UNICODE_TO_GBK[29010] := 16#83DC;
   // UNICODE_TO_GBK[29011] := 16#B2CB;
   // UNICODE_TO_GBK[29012] := 16#83DD;
   // UNICODE_TO_GBK[29013] := 16#DDC3;
   // UNICODE_TO_GBK[29014] := 16#83DE;
   // UNICODE_TO_GBK[29015] := 16#C797;
   // UNICODE_TO_GBK[29016] := 16#83DF;
   // UNICODE_TO_GBK[29017] := 16#DDCB;
   // UNICODE_TO_GBK[29018] := 16#83E0;
   // UNICODE_TO_GBK[29019] := 16#B2A4;
   // UNICODE_TO_GBK[29020] := 16#83E1;
   // UNICODE_TO_GBK[29021] := 16#DDD5;
   // UNICODE_TO_GBK[29022] := 16#83E2;
   // UNICODE_TO_GBK[29023] := 16#C798;
   // UNICODE_TO_GBK[29024] := 16#83E3;
   // UNICODE_TO_GBK[29025] := 16#C799;
   // UNICODE_TO_GBK[29026] := 16#83E4;
   // UNICODE_TO_GBK[29027] := 16#C79A;
   // UNICODE_TO_GBK[29028] := 16#83E5;
   // UNICODE_TO_GBK[29029] := 16#DDBE;
   // UNICODE_TO_GBK[29030] := 16#83E6;
   // UNICODE_TO_GBK[29031] := 16#C79B;
   // UNICODE_TO_GBK[29032] := 16#83E7;
   // UNICODE_TO_GBK[29033] := 16#C79C;
   // UNICODE_TO_GBK[29034] := 16#83E8;
   // UNICODE_TO_GBK[29035] := 16#C79D;
   // UNICODE_TO_GBK[29036] := 16#83E9;
   // UNICODE_TO_GBK[29037] := 16#C6D0;
   // UNICODE_TO_GBK[29038] := 16#83EA;
   // UNICODE_TO_GBK[29039] := 16#DDD0;
   // UNICODE_TO_GBK[29040] := 16#83EB;
   // UNICODE_TO_GBK[29041] := 16#C79E;
   // UNICODE_TO_GBK[29042] := 16#83EC;
   // UNICODE_TO_GBK[29043] := 16#C79F;
   // UNICODE_TO_GBK[29044] := 16#83ED;
   // UNICODE_TO_GBK[29045] := 16#C7A0;
   // UNICODE_TO_GBK[29046] := 16#83EE;
   // UNICODE_TO_GBK[29047] := 16#C840;
   // UNICODE_TO_GBK[29048] := 16#83EF;
   // UNICODE_TO_GBK[29049] := 16#C841;
   // UNICODE_TO_GBK[29050] := 16#83F0;
   // UNICODE_TO_GBK[29051] := 16#DDD4;
   // UNICODE_TO_GBK[29052] := 16#83F1;
   // UNICODE_TO_GBK[29053] := 16#C1E2;
   // UNICODE_TO_GBK[29054] := 16#83F2;
   // UNICODE_TO_GBK[29055] := 16#B7C6;
   // UNICODE_TO_GBK[29056] := 16#83F3;
   // UNICODE_TO_GBK[29057] := 16#C842;
   // UNICODE_TO_GBK[29058] := 16#83F4;
   // UNICODE_TO_GBK[29059] := 16#C843;
   // UNICODE_TO_GBK[29060] := 16#83F5;
   // UNICODE_TO_GBK[29061] := 16#C844;
   // UNICODE_TO_GBK[29062] := 16#83F6;
   // UNICODE_TO_GBK[29063] := 16#C845;
   // UNICODE_TO_GBK[29064] := 16#83F7;
   // UNICODE_TO_GBK[29065] := 16#C846;
   // UNICODE_TO_GBK[29066] := 16#83F8;
   // UNICODE_TO_GBK[29067] := 16#DDCE;
   // UNICODE_TO_GBK[29068] := 16#83F9;
   // UNICODE_TO_GBK[29069] := 16#DDCF;
   // UNICODE_TO_GBK[29070] := 16#83FA;
   // UNICODE_TO_GBK[29071] := 16#C847;
   // UNICODE_TO_GBK[29072] := 16#83FB;
   // UNICODE_TO_GBK[29073] := 16#C848;
   // UNICODE_TO_GBK[29074] := 16#83FC;
   // UNICODE_TO_GBK[29075] := 16#C849;
   // UNICODE_TO_GBK[29076] := 16#83FD;
   // UNICODE_TO_GBK[29077] := 16#DDC4;
   // UNICODE_TO_GBK[29078] := 16#83FE;
   // UNICODE_TO_GBK[29079] := 16#C84A;
   // UNICODE_TO_GBK[29080] := 16#83FF;
   // UNICODE_TO_GBK[29081] := 16#C84B;
   // UNICODE_TO_GBK[29082] := 16#8400;
   // UNICODE_TO_GBK[29083] := 16#C84C;
   // UNICODE_TO_GBK[29084] := 16#8401;
   // UNICODE_TO_GBK[29085] := 16#DDBD;
   // UNICODE_TO_GBK[29086] := 16#8402;
   // UNICODE_TO_GBK[29087] := 16#C84D;
   // UNICODE_TO_GBK[29088] := 16#8403;
   // UNICODE_TO_GBK[29089] := 16#DDCD;
   // UNICODE_TO_GBK[29090] := 16#8404;
   // UNICODE_TO_GBK[29091] := 16#CCD1;
   // UNICODE_TO_GBK[29092] := 16#8405;
   // UNICODE_TO_GBK[29093] := 16#C84E;
   // UNICODE_TO_GBK[29094] := 16#8406;
   // UNICODE_TO_GBK[29095] := 16#DDC9;
   // UNICODE_TO_GBK[29096] := 16#8407;
   // UNICODE_TO_GBK[29097] := 16#C84F;
   // UNICODE_TO_GBK[29098] := 16#8408;
   // UNICODE_TO_GBK[29099] := 16#C850;
   // UNICODE_TO_GBK[29100] := 16#8409;
   // UNICODE_TO_GBK[29101] := 16#C851;
   // UNICODE_TO_GBK[29102] := 16#840A;
   // UNICODE_TO_GBK[29103] := 16#C852;
   // UNICODE_TO_GBK[29104] := 16#840B;
   // UNICODE_TO_GBK[29105] := 16#DDC2;
   // UNICODE_TO_GBK[29106] := 16#840C;
   // UNICODE_TO_GBK[29107] := 16#C3C8;
   // UNICODE_TO_GBK[29108] := 16#840D;
   // UNICODE_TO_GBK[29109] := 16#C6BC;
   // UNICODE_TO_GBK[29110] := 16#840E;
   // UNICODE_TO_GBK[29111] := 16#CEAE;
   // UNICODE_TO_GBK[29112] := 16#840F;
   // UNICODE_TO_GBK[29113] := 16#DDCC;
   // UNICODE_TO_GBK[29114] := 16#8410;
   // UNICODE_TO_GBK[29115] := 16#C853;
   // UNICODE_TO_GBK[29116] := 16#8411;
   // UNICODE_TO_GBK[29117] := 16#DDC8;
   // UNICODE_TO_GBK[29118] := 16#8412;
   // UNICODE_TO_GBK[29119] := 16#C854;
   // UNICODE_TO_GBK[29120] := 16#8413;
   // UNICODE_TO_GBK[29121] := 16#C855;
   // UNICODE_TO_GBK[29122] := 16#8414;
   // UNICODE_TO_GBK[29123] := 16#C856;
   // UNICODE_TO_GBK[29124] := 16#8415;
   // UNICODE_TO_GBK[29125] := 16#C857;
   // UNICODE_TO_GBK[29126] := 16#8416;
   // UNICODE_TO_GBK[29127] := 16#C858;
   // UNICODE_TO_GBK[29128] := 16#8417;
   // UNICODE_TO_GBK[29129] := 16#C859;
   // UNICODE_TO_GBK[29130] := 16#8418;
   // UNICODE_TO_GBK[29131] := 16#DDC1;
   // UNICODE_TO_GBK[29132] := 16#8419;
   // UNICODE_TO_GBK[29133] := 16#C85A;
   // UNICODE_TO_GBK[29134] := 16#841A;
   // UNICODE_TO_GBK[29135] := 16#C85B;
   // UNICODE_TO_GBK[29136] := 16#841B;
   // UNICODE_TO_GBK[29137] := 16#C85C;
   // UNICODE_TO_GBK[29138] := 16#841C;
   // UNICODE_TO_GBK[29139] := 16#DDC6;
   // UNICODE_TO_GBK[29140] := 16#841D;
   // UNICODE_TO_GBK[29141] := 16#C2DC;
   // UNICODE_TO_GBK[29142] := 16#841E;
   // UNICODE_TO_GBK[29143] := 16#C85D;
   // UNICODE_TO_GBK[29144] := 16#841F;
   // UNICODE_TO_GBK[29145] := 16#C85E;
   // UNICODE_TO_GBK[29146] := 16#8420;
   // UNICODE_TO_GBK[29147] := 16#C85F;
   // UNICODE_TO_GBK[29148] := 16#8421;
   // UNICODE_TO_GBK[29149] := 16#C860;
   // UNICODE_TO_GBK[29150] := 16#8422;
   // UNICODE_TO_GBK[29151] := 16#C861;
   // UNICODE_TO_GBK[29152] := 16#8423;
   // UNICODE_TO_GBK[29153] := 16#C862;
   // UNICODE_TO_GBK[29154] := 16#8424;
   // UNICODE_TO_GBK[29155] := 16#D3A9;
   // UNICODE_TO_GBK[29156] := 16#8425;
   // UNICODE_TO_GBK[29157] := 16#D3AA;
   // UNICODE_TO_GBK[29158] := 16#8426;
   // UNICODE_TO_GBK[29159] := 16#DDD3;
   // UNICODE_TO_GBK[29160] := 16#8427;
   // UNICODE_TO_GBK[29161] := 16#CFF4;
   // UNICODE_TO_GBK[29162] := 16#8428;
   // UNICODE_TO_GBK[29163] := 16#C8F8;
   // UNICODE_TO_GBK[29164] := 16#8429;
   // UNICODE_TO_GBK[29165] := 16#C863;
   // UNICODE_TO_GBK[29166] := 16#842A;
   // UNICODE_TO_GBK[29167] := 16#C864;
   // UNICODE_TO_GBK[29168] := 16#842B;
   // UNICODE_TO_GBK[29169] := 16#C865;
   // UNICODE_TO_GBK[29170] := 16#842C;
   // UNICODE_TO_GBK[29171] := 16#C866;
   // UNICODE_TO_GBK[29172] := 16#842D;
   // UNICODE_TO_GBK[29173] := 16#C867;
   // UNICODE_TO_GBK[29174] := 16#842E;
   // UNICODE_TO_GBK[29175] := 16#C868;
   // UNICODE_TO_GBK[29176] := 16#842F;
   // UNICODE_TO_GBK[29177] := 16#C869;
   // UNICODE_TO_GBK[29178] := 16#8430;
   // UNICODE_TO_GBK[29179] := 16#C86A;
   // UNICODE_TO_GBK[29180] := 16#8431;
   // UNICODE_TO_GBK[29181] := 16#DDE6;
   // UNICODE_TO_GBK[29182] := 16#8432;
   // UNICODE_TO_GBK[29183] := 16#C86B;
   // UNICODE_TO_GBK[29184] := 16#8433;
   // UNICODE_TO_GBK[29185] := 16#C86C;
   // UNICODE_TO_GBK[29186] := 16#8434;
   // UNICODE_TO_GBK[29187] := 16#C86D;
   // UNICODE_TO_GBK[29188] := 16#8435;
   // UNICODE_TO_GBK[29189] := 16#C86E;
   // UNICODE_TO_GBK[29190] := 16#8436;
   // UNICODE_TO_GBK[29191] := 16#C86F;
   // UNICODE_TO_GBK[29192] := 16#8437;
   // UNICODE_TO_GBK[29193] := 16#C870;
   // UNICODE_TO_GBK[29194] := 16#8438;
   // UNICODE_TO_GBK[29195] := 16#DDC7;
   // UNICODE_TO_GBK[29196] := 16#8439;
   // UNICODE_TO_GBK[29197] := 16#C871;
   // UNICODE_TO_GBK[29198] := 16#843A;
   // UNICODE_TO_GBK[29199] := 16#C872;
   // UNICODE_TO_GBK[29200] := 16#843B;
   // UNICODE_TO_GBK[29201] := 16#C873;
   // UNICODE_TO_GBK[29202] := 16#843C;
   // UNICODE_TO_GBK[29203] := 16#DDE0;
   // UNICODE_TO_GBK[29204] := 16#843D;
   // UNICODE_TO_GBK[29205] := 16#C2E4;
   // UNICODE_TO_GBK[29206] := 16#843E;
   // UNICODE_TO_GBK[29207] := 16#C874;
   // UNICODE_TO_GBK[29208] := 16#843F;
   // UNICODE_TO_GBK[29209] := 16#C875;
   // UNICODE_TO_GBK[29210] := 16#8440;
   // UNICODE_TO_GBK[29211] := 16#C876;
   // UNICODE_TO_GBK[29212] := 16#8441;
   // UNICODE_TO_GBK[29213] := 16#C877;
   // UNICODE_TO_GBK[29214] := 16#8442;
   // UNICODE_TO_GBK[29215] := 16#C878;
   // UNICODE_TO_GBK[29216] := 16#8443;
   // UNICODE_TO_GBK[29217] := 16#C879;
   // UNICODE_TO_GBK[29218] := 16#8444;
   // UNICODE_TO_GBK[29219] := 16#C87A;
   // UNICODE_TO_GBK[29220] := 16#8445;
   // UNICODE_TO_GBK[29221] := 16#C87B;
   // UNICODE_TO_GBK[29222] := 16#8446;
   // UNICODE_TO_GBK[29223] := 16#DDE1;
   // UNICODE_TO_GBK[29224] := 16#8447;
   // UNICODE_TO_GBK[29225] := 16#C87C;
   // UNICODE_TO_GBK[29226] := 16#8448;
   // UNICODE_TO_GBK[29227] := 16#C87D;
   // UNICODE_TO_GBK[29228] := 16#8449;
   // UNICODE_TO_GBK[29229] := 16#C87E;
   // UNICODE_TO_GBK[29230] := 16#844A;
   // UNICODE_TO_GBK[29231] := 16#C880;
   // UNICODE_TO_GBK[29232] := 16#844B;
   // UNICODE_TO_GBK[29233] := 16#C881;
   // UNICODE_TO_GBK[29234] := 16#844C;
   // UNICODE_TO_GBK[29235] := 16#C882;
   // UNICODE_TO_GBK[29236] := 16#844D;
   // UNICODE_TO_GBK[29237] := 16#C883;
   // UNICODE_TO_GBK[29238] := 16#844E;
   // UNICODE_TO_GBK[29239] := 16#C884;
   // UNICODE_TO_GBK[29240] := 16#844F;
   // UNICODE_TO_GBK[29241] := 16#C885;
   // UNICODE_TO_GBK[29242] := 16#8450;
   // UNICODE_TO_GBK[29243] := 16#C886;
   // UNICODE_TO_GBK[29244] := 16#8451;
   // UNICODE_TO_GBK[29245] := 16#DDD7;
   // UNICODE_TO_GBK[29246] := 16#8452;
   // UNICODE_TO_GBK[29247] := 16#C887;
   // UNICODE_TO_GBK[29248] := 16#8453;
   // UNICODE_TO_GBK[29249] := 16#C888;
   // UNICODE_TO_GBK[29250] := 16#8454;
   // UNICODE_TO_GBK[29251] := 16#C889;
   // UNICODE_TO_GBK[29252] := 16#8455;
   // UNICODE_TO_GBK[29253] := 16#C88A;
   // UNICODE_TO_GBK[29254] := 16#8456;
   // UNICODE_TO_GBK[29255] := 16#C88B;
   // UNICODE_TO_GBK[29256] := 16#8457;
   // UNICODE_TO_GBK[29257] := 16#D6F8;
   // UNICODE_TO_GBK[29258] := 16#8458;
   // UNICODE_TO_GBK[29259] := 16#C88C;
   // UNICODE_TO_GBK[29260] := 16#8459;
   // UNICODE_TO_GBK[29261] := 16#DDD9;
   // UNICODE_TO_GBK[29262] := 16#845A;
   // UNICODE_TO_GBK[29263] := 16#DDD8;
   // UNICODE_TO_GBK[29264] := 16#845B;
   // UNICODE_TO_GBK[29265] := 16#B8F0;
   // UNICODE_TO_GBK[29266] := 16#845C;
   // UNICODE_TO_GBK[29267] := 16#DDD6;
   // UNICODE_TO_GBK[29268] := 16#845D;
   // UNICODE_TO_GBK[29269] := 16#C88D;
   // UNICODE_TO_GBK[29270] := 16#845E;
   // UNICODE_TO_GBK[29271] := 16#C88E;
   // UNICODE_TO_GBK[29272] := 16#845F;
   // UNICODE_TO_GBK[29273] := 16#C88F;
   // UNICODE_TO_GBK[29274] := 16#8460;
   // UNICODE_TO_GBK[29275] := 16#C890;
   // UNICODE_TO_GBK[29276] := 16#8461;
   // UNICODE_TO_GBK[29277] := 16#C6CF;
   // UNICODE_TO_GBK[29278] := 16#8462;
   // UNICODE_TO_GBK[29279] := 16#C891;
   // UNICODE_TO_GBK[29280] := 16#8463;
   // UNICODE_TO_GBK[29281] := 16#B6AD;
   // UNICODE_TO_GBK[29282] := 16#8464;
   // UNICODE_TO_GBK[29283] := 16#C892;
   // UNICODE_TO_GBK[29284] := 16#8465;
   // UNICODE_TO_GBK[29285] := 16#C893;
   // UNICODE_TO_GBK[29286] := 16#8466;
   // UNICODE_TO_GBK[29287] := 16#C894;
   // UNICODE_TO_GBK[29288] := 16#8467;
   // UNICODE_TO_GBK[29289] := 16#C895;
   // UNICODE_TO_GBK[29290] := 16#8468;
   // UNICODE_TO_GBK[29291] := 16#C896;
   // UNICODE_TO_GBK[29292] := 16#8469;
   // UNICODE_TO_GBK[29293] := 16#DDE2;
   // UNICODE_TO_GBK[29294] := 16#846A;
   // UNICODE_TO_GBK[29295] := 16#C897;
   // UNICODE_TO_GBK[29296] := 16#846B;
   // UNICODE_TO_GBK[29297] := 16#BAF9;
   // UNICODE_TO_GBK[29298] := 16#846C;
   // UNICODE_TO_GBK[29299] := 16#D4E1;
   // UNICODE_TO_GBK[29300] := 16#846D;
   // UNICODE_TO_GBK[29301] := 16#DDE7;
   // UNICODE_TO_GBK[29302] := 16#846E;
   // UNICODE_TO_GBK[29303] := 16#C898;
   // UNICODE_TO_GBK[29304] := 16#846F;
   // UNICODE_TO_GBK[29305] := 16#C899;
   // UNICODE_TO_GBK[29306] := 16#8470;
   // UNICODE_TO_GBK[29307] := 16#C89A;
   // UNICODE_TO_GBK[29308] := 16#8471;
   // UNICODE_TO_GBK[29309] := 16#B4D0;
   // UNICODE_TO_GBK[29310] := 16#8472;
   // UNICODE_TO_GBK[29311] := 16#C89B;
   // UNICODE_TO_GBK[29312] := 16#8473;
   // UNICODE_TO_GBK[29313] := 16#DDDA;
   // UNICODE_TO_GBK[29314] := 16#8474;
   // UNICODE_TO_GBK[29315] := 16#C89C;
   // UNICODE_TO_GBK[29316] := 16#8475;
   // UNICODE_TO_GBK[29317] := 16#BFFB;
   // UNICODE_TO_GBK[29318] := 16#8476;
   // UNICODE_TO_GBK[29319] := 16#DDE3;
   // UNICODE_TO_GBK[29320] := 16#8477;
   // UNICODE_TO_GBK[29321] := 16#C89D;
   // UNICODE_TO_GBK[29322] := 16#8478;
   // UNICODE_TO_GBK[29323] := 16#DDDF;
   // UNICODE_TO_GBK[29324] := 16#8479;
   // UNICODE_TO_GBK[29325] := 16#C89E;
   // UNICODE_TO_GBK[29326] := 16#847A;
   // UNICODE_TO_GBK[29327] := 16#DDDD;
   // UNICODE_TO_GBK[29328] := 16#847B;
   // UNICODE_TO_GBK[29329] := 16#C89F;
   // UNICODE_TO_GBK[29330] := 16#847C;
   // UNICODE_TO_GBK[29331] := 16#C8A0;
   // UNICODE_TO_GBK[29332] := 16#847D;
   // UNICODE_TO_GBK[29333] := 16#C940;
   // UNICODE_TO_GBK[29334] := 16#847E;
   // UNICODE_TO_GBK[29335] := 16#C941;
   // UNICODE_TO_GBK[29336] := 16#847F;
   // UNICODE_TO_GBK[29337] := 16#C942;
   // UNICODE_TO_GBK[29338] := 16#8480;
   // UNICODE_TO_GBK[29339] := 16#C943;
   // UNICODE_TO_GBK[29340] := 16#8481;
   // UNICODE_TO_GBK[29341] := 16#C944;
   // UNICODE_TO_GBK[29342] := 16#8482;
   // UNICODE_TO_GBK[29343] := 16#B5D9;
   // UNICODE_TO_GBK[29344] := 16#8483;
   // UNICODE_TO_GBK[29345] := 16#C945;
   // UNICODE_TO_GBK[29346] := 16#8484;
   // UNICODE_TO_GBK[29347] := 16#C946;
   // UNICODE_TO_GBK[29348] := 16#8485;
   // UNICODE_TO_GBK[29349] := 16#C947;
   // UNICODE_TO_GBK[29350] := 16#8486;
   // UNICODE_TO_GBK[29351] := 16#C948;
   // UNICODE_TO_GBK[29352] := 16#8487;
   // UNICODE_TO_GBK[29353] := 16#DDDB;
   // UNICODE_TO_GBK[29354] := 16#8488;
   // UNICODE_TO_GBK[29355] := 16#DDDC;
   // UNICODE_TO_GBK[29356] := 16#8489;
   // UNICODE_TO_GBK[29357] := 16#DDDE;
   // UNICODE_TO_GBK[29358] := 16#848A;
   // UNICODE_TO_GBK[29359] := 16#C949;
   // UNICODE_TO_GBK[29360] := 16#848B;
   // UNICODE_TO_GBK[29361] := 16#BDAF;
   // UNICODE_TO_GBK[29362] := 16#848C;
   // UNICODE_TO_GBK[29363] := 16#DDE4;
   // UNICODE_TO_GBK[29364] := 16#848D;
   // UNICODE_TO_GBK[29365] := 16#C94A;
   // UNICODE_TO_GBK[29366] := 16#848E;
   // UNICODE_TO_GBK[29367] := 16#DDE5;
   // UNICODE_TO_GBK[29368] := 16#848F;
   // UNICODE_TO_GBK[29369] := 16#C94B;
   // UNICODE_TO_GBK[29370] := 16#8490;
   // UNICODE_TO_GBK[29371] := 16#C94C;
   // UNICODE_TO_GBK[29372] := 16#8491;
   // UNICODE_TO_GBK[29373] := 16#C94D;
   // UNICODE_TO_GBK[29374] := 16#8492;
   // UNICODE_TO_GBK[29375] := 16#C94E;
   // UNICODE_TO_GBK[29376] := 16#8493;
   // UNICODE_TO_GBK[29377] := 16#C94F;
   // UNICODE_TO_GBK[29378] := 16#8494;
   // UNICODE_TO_GBK[29379] := 16#C950;
   // UNICODE_TO_GBK[29380] := 16#8495;
   // UNICODE_TO_GBK[29381] := 16#C951;
   // UNICODE_TO_GBK[29382] := 16#8496;
   // UNICODE_TO_GBK[29383] := 16#C952;
   // UNICODE_TO_GBK[29384] := 16#8497;
   // UNICODE_TO_GBK[29385] := 16#DDF5;
   // UNICODE_TO_GBK[29386] := 16#8498;
   // UNICODE_TO_GBK[29387] := 16#C953;
   // UNICODE_TO_GBK[29388] := 16#8499;
   // UNICODE_TO_GBK[29389] := 16#C3C9;
   // UNICODE_TO_GBK[29390] := 16#849A;
   // UNICODE_TO_GBK[29391] := 16#C954;
   // UNICODE_TO_GBK[29392] := 16#849B;
   // UNICODE_TO_GBK[29393] := 16#C955;
   // UNICODE_TO_GBK[29394] := 16#849C;
   // UNICODE_TO_GBK[29395] := 16#CBE2;
   // UNICODE_TO_GBK[29396] := 16#849D;
   // UNICODE_TO_GBK[29397] := 16#C956;
   // UNICODE_TO_GBK[29398] := 16#849E;
   // UNICODE_TO_GBK[29399] := 16#C957;
   // UNICODE_TO_GBK[29400] := 16#849F;
   // UNICODE_TO_GBK[29401] := 16#C958;
   // UNICODE_TO_GBK[29402] := 16#84A0;
   // UNICODE_TO_GBK[29403] := 16#C959;
   // UNICODE_TO_GBK[29404] := 16#84A1;
   // UNICODE_TO_GBK[29405] := 16#DDF2;
   // UNICODE_TO_GBK[29406] := 16#84A2;
   // UNICODE_TO_GBK[29407] := 16#C95A;
   // UNICODE_TO_GBK[29408] := 16#84A3;
   // UNICODE_TO_GBK[29409] := 16#C95B;
   // UNICODE_TO_GBK[29410] := 16#84A4;
   // UNICODE_TO_GBK[29411] := 16#C95C;
   // UNICODE_TO_GBK[29412] := 16#84A5;
   // UNICODE_TO_GBK[29413] := 16#C95D;
   // UNICODE_TO_GBK[29414] := 16#84A6;
   // UNICODE_TO_GBK[29415] := 16#C95E;
   // UNICODE_TO_GBK[29416] := 16#84A7;
   // UNICODE_TO_GBK[29417] := 16#C95F;
   // UNICODE_TO_GBK[29418] := 16#84A8;
   // UNICODE_TO_GBK[29419] := 16#C960;
   // UNICODE_TO_GBK[29420] := 16#84A9;
   // UNICODE_TO_GBK[29421] := 16#C961;
   // UNICODE_TO_GBK[29422] := 16#84AA;
   // UNICODE_TO_GBK[29423] := 16#C962;
   // UNICODE_TO_GBK[29424] := 16#84AB;
   // UNICODE_TO_GBK[29425] := 16#C963;
   // UNICODE_TO_GBK[29426] := 16#84AC;
   // UNICODE_TO_GBK[29427] := 16#C964;
   // UNICODE_TO_GBK[29428] := 16#84AD;
   // UNICODE_TO_GBK[29429] := 16#C965;
   // UNICODE_TO_GBK[29430] := 16#84AE;
   // UNICODE_TO_GBK[29431] := 16#C966;
   // UNICODE_TO_GBK[29432] := 16#84AF;
   // UNICODE_TO_GBK[29433] := 16#D8E1;
   // UNICODE_TO_GBK[29434] := 16#84B0;
   // UNICODE_TO_GBK[29435] := 16#C967;
   // UNICODE_TO_GBK[29436] := 16#84B1;
   // UNICODE_TO_GBK[29437] := 16#C968;
   // UNICODE_TO_GBK[29438] := 16#84B2;
   // UNICODE_TO_GBK[29439] := 16#C6D1;
   // UNICODE_TO_GBK[29440] := 16#84B3;
   // UNICODE_TO_GBK[29441] := 16#C969;
   // UNICODE_TO_GBK[29442] := 16#84B4;
   // UNICODE_TO_GBK[29443] := 16#DDF4;
   // UNICODE_TO_GBK[29444] := 16#84B5;
   // UNICODE_TO_GBK[29445] := 16#C96A;
   // UNICODE_TO_GBK[29446] := 16#84B6;
   // UNICODE_TO_GBK[29447] := 16#C96B;
   // UNICODE_TO_GBK[29448] := 16#84B7;
   // UNICODE_TO_GBK[29449] := 16#C96C;
   // UNICODE_TO_GBK[29450] := 16#84B8;
   // UNICODE_TO_GBK[29451] := 16#D5F4;
   // UNICODE_TO_GBK[29452] := 16#84B9;
   // UNICODE_TO_GBK[29453] := 16#DDF3;
   // UNICODE_TO_GBK[29454] := 16#84BA;
   // UNICODE_TO_GBK[29455] := 16#DDF0;
   // UNICODE_TO_GBK[29456] := 16#84BB;
   // UNICODE_TO_GBK[29457] := 16#C96D;
   // UNICODE_TO_GBK[29458] := 16#84BC;
   // UNICODE_TO_GBK[29459] := 16#C96E;
   // UNICODE_TO_GBK[29460] := 16#84BD;
   // UNICODE_TO_GBK[29461] := 16#DDEC;
   // UNICODE_TO_GBK[29462] := 16#84BE;
   // UNICODE_TO_GBK[29463] := 16#C96F;
   // UNICODE_TO_GBK[29464] := 16#84BF;
   // UNICODE_TO_GBK[29465] := 16#DDEF;
   // UNICODE_TO_GBK[29466] := 16#84C0;
   // UNICODE_TO_GBK[29467] := 16#C970;
   // UNICODE_TO_GBK[29468] := 16#84C1;
   // UNICODE_TO_GBK[29469] := 16#DDE8;
   // UNICODE_TO_GBK[29470] := 16#84C2;
   // UNICODE_TO_GBK[29471] := 16#C971;
   // UNICODE_TO_GBK[29472] := 16#84C3;
   // UNICODE_TO_GBK[29473] := 16#C972;
   // UNICODE_TO_GBK[29474] := 16#84C4;
   // UNICODE_TO_GBK[29475] := 16#D0EE;
   // UNICODE_TO_GBK[29476] := 16#84C5;
   // UNICODE_TO_GBK[29477] := 16#C973;
   // UNICODE_TO_GBK[29478] := 16#84C6;
   // UNICODE_TO_GBK[29479] := 16#C974;
   // UNICODE_TO_GBK[29480] := 16#84C7;
   // UNICODE_TO_GBK[29481] := 16#C975;
   // UNICODE_TO_GBK[29482] := 16#84C8;
   // UNICODE_TO_GBK[29483] := 16#C976;
   // UNICODE_TO_GBK[29484] := 16#84C9;
   // UNICODE_TO_GBK[29485] := 16#C8D8;
   // UNICODE_TO_GBK[29486] := 16#84CA;
   // UNICODE_TO_GBK[29487] := 16#DDEE;
   // UNICODE_TO_GBK[29488] := 16#84CB;
   // UNICODE_TO_GBK[29489] := 16#C977;
   // UNICODE_TO_GBK[29490] := 16#84CC;
   // UNICODE_TO_GBK[29491] := 16#C978;
   // UNICODE_TO_GBK[29492] := 16#84CD;
   // UNICODE_TO_GBK[29493] := 16#DDE9;
   // UNICODE_TO_GBK[29494] := 16#84CE;
   // UNICODE_TO_GBK[29495] := 16#C979;
   // UNICODE_TO_GBK[29496] := 16#84CF;
   // UNICODE_TO_GBK[29497] := 16#C97A;
   // UNICODE_TO_GBK[29498] := 16#84D0;
   // UNICODE_TO_GBK[29499] := 16#DDEA;
   // UNICODE_TO_GBK[29500] := 16#84D1;
   // UNICODE_TO_GBK[29501] := 16#CBF2;
   // UNICODE_TO_GBK[29502] := 16#84D2;
   // UNICODE_TO_GBK[29503] := 16#C97B;
   // UNICODE_TO_GBK[29504] := 16#84D3;
   // UNICODE_TO_GBK[29505] := 16#DDED;
   // UNICODE_TO_GBK[29506] := 16#84D4;
   // UNICODE_TO_GBK[29507] := 16#C97C;
   // UNICODE_TO_GBK[29508] := 16#84D5;
   // UNICODE_TO_GBK[29509] := 16#C97D;
   // UNICODE_TO_GBK[29510] := 16#84D6;
   // UNICODE_TO_GBK[29511] := 16#B1CD;
   // UNICODE_TO_GBK[29512] := 16#84D7;
   // UNICODE_TO_GBK[29513] := 16#C97E;
   // UNICODE_TO_GBK[29514] := 16#84D8;
   // UNICODE_TO_GBK[29515] := 16#C980;
   // UNICODE_TO_GBK[29516] := 16#84D9;
   // UNICODE_TO_GBK[29517] := 16#C981;
   // UNICODE_TO_GBK[29518] := 16#84DA;
   // UNICODE_TO_GBK[29519] := 16#C982;
   // UNICODE_TO_GBK[29520] := 16#84DB;
   // UNICODE_TO_GBK[29521] := 16#C983;
   // UNICODE_TO_GBK[29522] := 16#84DC;
   // UNICODE_TO_GBK[29523] := 16#C984;
   // UNICODE_TO_GBK[29524] := 16#84DD;
   // UNICODE_TO_GBK[29525] := 16#C0B6;
   // UNICODE_TO_GBK[29526] := 16#84DE;
   // UNICODE_TO_GBK[29527] := 16#C985;
   // UNICODE_TO_GBK[29528] := 16#84DF;
   // UNICODE_TO_GBK[29529] := 16#BCBB;
   // UNICODE_TO_GBK[29530] := 16#84E0;
   // UNICODE_TO_GBK[29531] := 16#DDF1;
   // UNICODE_TO_GBK[29532] := 16#84E1;
   // UNICODE_TO_GBK[29533] := 16#C986;
   // UNICODE_TO_GBK[29534] := 16#84E2;
   // UNICODE_TO_GBK[29535] := 16#C987;
   // UNICODE_TO_GBK[29536] := 16#84E3;
   // UNICODE_TO_GBK[29537] := 16#DDF7;
   // UNICODE_TO_GBK[29538] := 16#84E4;
   // UNICODE_TO_GBK[29539] := 16#C988;
   // UNICODE_TO_GBK[29540] := 16#84E5;
   // UNICODE_TO_GBK[29541] := 16#DDF6;
   // UNICODE_TO_GBK[29542] := 16#84E6;
   // UNICODE_TO_GBK[29543] := 16#DDEB;
   // UNICODE_TO_GBK[29544] := 16#84E7;
   // UNICODE_TO_GBK[29545] := 16#C989;
   // UNICODE_TO_GBK[29546] := 16#84E8;
   // UNICODE_TO_GBK[29547] := 16#C98A;
   // UNICODE_TO_GBK[29548] := 16#84E9;
   // UNICODE_TO_GBK[29549] := 16#C98B;
   // UNICODE_TO_GBK[29550] := 16#84EA;
   // UNICODE_TO_GBK[29551] := 16#C98C;
   // UNICODE_TO_GBK[29552] := 16#84EB;
   // UNICODE_TO_GBK[29553] := 16#C98D;
   // UNICODE_TO_GBK[29554] := 16#84EC;
   // UNICODE_TO_GBK[29555] := 16#C5EE;
   // UNICODE_TO_GBK[29556] := 16#84ED;
   // UNICODE_TO_GBK[29557] := 16#C98E;
   // UNICODE_TO_GBK[29558] := 16#84EE;
   // UNICODE_TO_GBK[29559] := 16#C98F;
   // UNICODE_TO_GBK[29560] := 16#84EF;
   // UNICODE_TO_GBK[29561] := 16#C990;
   // UNICODE_TO_GBK[29562] := 16#84F0;
   // UNICODE_TO_GBK[29563] := 16#DDFB;
   // UNICODE_TO_GBK[29564] := 16#84F1;
   // UNICODE_TO_GBK[29565] := 16#C991;
   // UNICODE_TO_GBK[29566] := 16#84F2;
   // UNICODE_TO_GBK[29567] := 16#C992;
   // UNICODE_TO_GBK[29568] := 16#84F3;
   // UNICODE_TO_GBK[29569] := 16#C993;
   // UNICODE_TO_GBK[29570] := 16#84F4;
   // UNICODE_TO_GBK[29571] := 16#C994;
   // UNICODE_TO_GBK[29572] := 16#84F5;
   // UNICODE_TO_GBK[29573] := 16#C995;
   // UNICODE_TO_GBK[29574] := 16#84F6;
   // UNICODE_TO_GBK[29575] := 16#C996;
   // UNICODE_TO_GBK[29576] := 16#84F7;
   // UNICODE_TO_GBK[29577] := 16#C997;
   // UNICODE_TO_GBK[29578] := 16#84F8;
   // UNICODE_TO_GBK[29579] := 16#C998;
   // UNICODE_TO_GBK[29580] := 16#84F9;
   // UNICODE_TO_GBK[29581] := 16#C999;
   // UNICODE_TO_GBK[29582] := 16#84FA;
   // UNICODE_TO_GBK[29583] := 16#C99A;
   // UNICODE_TO_GBK[29584] := 16#84FB;
   // UNICODE_TO_GBK[29585] := 16#C99B;
   // UNICODE_TO_GBK[29586] := 16#84FC;
   // UNICODE_TO_GBK[29587] := 16#DEA4;
   // UNICODE_TO_GBK[29588] := 16#84FD;
   // UNICODE_TO_GBK[29589] := 16#C99C;
   // UNICODE_TO_GBK[29590] := 16#84FE;
   // UNICODE_TO_GBK[29591] := 16#C99D;
   // UNICODE_TO_GBK[29592] := 16#84FF;
   // UNICODE_TO_GBK[29593] := 16#DEA3;
   // UNICODE_TO_GBK[29594] := 16#8500;
   // UNICODE_TO_GBK[29595] := 16#C99E;
   // UNICODE_TO_GBK[29596] := 16#8501;
   // UNICODE_TO_GBK[29597] := 16#C99F;
   // UNICODE_TO_GBK[29598] := 16#8502;
   // UNICODE_TO_GBK[29599] := 16#C9A0;
   // UNICODE_TO_GBK[29600] := 16#8503;
   // UNICODE_TO_GBK[29601] := 16#CA40;
   // UNICODE_TO_GBK[29602] := 16#8504;
   // UNICODE_TO_GBK[29603] := 16#CA41;
   // UNICODE_TO_GBK[29604] := 16#8505;
   // UNICODE_TO_GBK[29605] := 16#CA42;
   // UNICODE_TO_GBK[29606] := 16#8506;
   // UNICODE_TO_GBK[29607] := 16#CA43;
   // UNICODE_TO_GBK[29608] := 16#8507;
   // UNICODE_TO_GBK[29609] := 16#CA44;
   // UNICODE_TO_GBK[29610] := 16#8508;
   // UNICODE_TO_GBK[29611] := 16#CA45;
   // UNICODE_TO_GBK[29612] := 16#8509;
   // UNICODE_TO_GBK[29613] := 16#CA46;
   // UNICODE_TO_GBK[29614] := 16#850A;
   // UNICODE_TO_GBK[29615] := 16#CA47;
   // UNICODE_TO_GBK[29616] := 16#850B;
   // UNICODE_TO_GBK[29617] := 16#CA48;
   // UNICODE_TO_GBK[29618] := 16#850C;
   // UNICODE_TO_GBK[29619] := 16#DDF8;
   // UNICODE_TO_GBK[29620] := 16#850D;
   // UNICODE_TO_GBK[29621] := 16#CA49;
   // UNICODE_TO_GBK[29622] := 16#850E;
   // UNICODE_TO_GBK[29623] := 16#CA4A;
   // UNICODE_TO_GBK[29624] := 16#850F;
   // UNICODE_TO_GBK[29625] := 16#CA4B;
   // UNICODE_TO_GBK[29626] := 16#8510;
   // UNICODE_TO_GBK[29627] := 16#CA4C;
   // UNICODE_TO_GBK[29628] := 16#8511;
   // UNICODE_TO_GBK[29629] := 16#C3EF;
   // UNICODE_TO_GBK[29630] := 16#8512;
   // UNICODE_TO_GBK[29631] := 16#CA4D;
   // UNICODE_TO_GBK[29632] := 16#8513;
   // UNICODE_TO_GBK[29633] := 16#C2FB;
   // UNICODE_TO_GBK[29634] := 16#8514;
   // UNICODE_TO_GBK[29635] := 16#CA4E;
   // UNICODE_TO_GBK[29636] := 16#8515;
   // UNICODE_TO_GBK[29637] := 16#CA4F;
   // UNICODE_TO_GBK[29638] := 16#8516;
   // UNICODE_TO_GBK[29639] := 16#CA50;
   // UNICODE_TO_GBK[29640] := 16#8517;
   // UNICODE_TO_GBK[29641] := 16#D5E1;
   // UNICODE_TO_GBK[29642] := 16#8518;
   // UNICODE_TO_GBK[29643] := 16#CA51;
   // UNICODE_TO_GBK[29644] := 16#8519;
   // UNICODE_TO_GBK[29645] := 16#CA52;
   // UNICODE_TO_GBK[29646] := 16#851A;
   // UNICODE_TO_GBK[29647] := 16#CEB5;
   // UNICODE_TO_GBK[29648] := 16#851B;
   // UNICODE_TO_GBK[29649] := 16#CA53;
   // UNICODE_TO_GBK[29650] := 16#851C;
   // UNICODE_TO_GBK[29651] := 16#CA54;
   // UNICODE_TO_GBK[29652] := 16#851D;
   // UNICODE_TO_GBK[29653] := 16#CA55;
   // UNICODE_TO_GBK[29654] := 16#851E;
   // UNICODE_TO_GBK[29655] := 16#CA56;
   // UNICODE_TO_GBK[29656] := 16#851F;
   // UNICODE_TO_GBK[29657] := 16#DDFD;
   // UNICODE_TO_GBK[29658] := 16#8520;
   // UNICODE_TO_GBK[29659] := 16#CA57;
   // UNICODE_TO_GBK[29660] := 16#8521;
   // UNICODE_TO_GBK[29661] := 16#B2CC;
   // UNICODE_TO_GBK[29662] := 16#8522;
   // UNICODE_TO_GBK[29663] := 16#CA58;
   // UNICODE_TO_GBK[29664] := 16#8523;
   // UNICODE_TO_GBK[29665] := 16#CA59;
   // UNICODE_TO_GBK[29666] := 16#8524;
   // UNICODE_TO_GBK[29667] := 16#CA5A;
   // UNICODE_TO_GBK[29668] := 16#8525;
   // UNICODE_TO_GBK[29669] := 16#CA5B;
   // UNICODE_TO_GBK[29670] := 16#8526;
   // UNICODE_TO_GBK[29671] := 16#CA5C;
   // UNICODE_TO_GBK[29672] := 16#8527;
   // UNICODE_TO_GBK[29673] := 16#CA5D;
   // UNICODE_TO_GBK[29674] := 16#8528;
   // UNICODE_TO_GBK[29675] := 16#CA5E;
   // UNICODE_TO_GBK[29676] := 16#8529;
   // UNICODE_TO_GBK[29677] := 16#CA5F;
   // UNICODE_TO_GBK[29678] := 16#852A;
   // UNICODE_TO_GBK[29679] := 16#CA60;
   // UNICODE_TO_GBK[29680] := 16#852B;
   // UNICODE_TO_GBK[29681] := 16#C4E8;
   // UNICODE_TO_GBK[29682] := 16#852C;
   // UNICODE_TO_GBK[29683] := 16#CADF;
   // UNICODE_TO_GBK[29684] := 16#852D;
   // UNICODE_TO_GBK[29685] := 16#CA61;
   // UNICODE_TO_GBK[29686] := 16#852E;
   // UNICODE_TO_GBK[29687] := 16#CA62;
   // UNICODE_TO_GBK[29688] := 16#852F;
   // UNICODE_TO_GBK[29689] := 16#CA63;
   // UNICODE_TO_GBK[29690] := 16#8530;
   // UNICODE_TO_GBK[29691] := 16#CA64;
   // UNICODE_TO_GBK[29692] := 16#8531;
   // UNICODE_TO_GBK[29693] := 16#CA65;
   // UNICODE_TO_GBK[29694] := 16#8532;
   // UNICODE_TO_GBK[29695] := 16#CA66;
   // UNICODE_TO_GBK[29696] := 16#8533;
   // UNICODE_TO_GBK[29697] := 16#CA67;
   // UNICODE_TO_GBK[29698] := 16#8534;
   // UNICODE_TO_GBK[29699] := 16#CA68;
   // UNICODE_TO_GBK[29700] := 16#8535;
   // UNICODE_TO_GBK[29701] := 16#CA69;
   // UNICODE_TO_GBK[29702] := 16#8536;
   // UNICODE_TO_GBK[29703] := 16#CA6A;
   // UNICODE_TO_GBK[29704] := 16#8537;
   // UNICODE_TO_GBK[29705] := 16#C7BE;
   // UNICODE_TO_GBK[29706] := 16#8538;
   // UNICODE_TO_GBK[29707] := 16#DDFA;
   // UNICODE_TO_GBK[29708] := 16#8539;
   // UNICODE_TO_GBK[29709] := 16#DDFC;
   // UNICODE_TO_GBK[29710] := 16#853A;
   // UNICODE_TO_GBK[29711] := 16#DDFE;
   // UNICODE_TO_GBK[29712] := 16#853B;
   // UNICODE_TO_GBK[29713] := 16#DEA2;
   // UNICODE_TO_GBK[29714] := 16#853C;
   // UNICODE_TO_GBK[29715] := 16#B0AA;
   // UNICODE_TO_GBK[29716] := 16#853D;
   // UNICODE_TO_GBK[29717] := 16#B1CE;
   // UNICODE_TO_GBK[29718] := 16#853E;
   // UNICODE_TO_GBK[29719] := 16#CA6B;
   // UNICODE_TO_GBK[29720] := 16#853F;
   // UNICODE_TO_GBK[29721] := 16#CA6C;
   // UNICODE_TO_GBK[29722] := 16#8540;
   // UNICODE_TO_GBK[29723] := 16#CA6D;
   // UNICODE_TO_GBK[29724] := 16#8541;
   // UNICODE_TO_GBK[29725] := 16#CA6E;
   // UNICODE_TO_GBK[29726] := 16#8542;
   // UNICODE_TO_GBK[29727] := 16#CA6F;
   // UNICODE_TO_GBK[29728] := 16#8543;
   // UNICODE_TO_GBK[29729] := 16#DEAC;
   // UNICODE_TO_GBK[29730] := 16#8544;
   // UNICODE_TO_GBK[29731] := 16#CA70;
   // UNICODE_TO_GBK[29732] := 16#8545;
   // UNICODE_TO_GBK[29733] := 16#CA71;
   // UNICODE_TO_GBK[29734] := 16#8546;
   // UNICODE_TO_GBK[29735] := 16#CA72;
   // UNICODE_TO_GBK[29736] := 16#8547;
   // UNICODE_TO_GBK[29737] := 16#CA73;
   // UNICODE_TO_GBK[29738] := 16#8548;
   // UNICODE_TO_GBK[29739] := 16#DEA6;
   // UNICODE_TO_GBK[29740] := 16#8549;
   // UNICODE_TO_GBK[29741] := 16#BDB6;
   // UNICODE_TO_GBK[29742] := 16#854A;
   // UNICODE_TO_GBK[29743] := 16#C8EF;
   // UNICODE_TO_GBK[29744] := 16#854B;
   // UNICODE_TO_GBK[29745] := 16#CA74;
   // UNICODE_TO_GBK[29746] := 16#854C;
   // UNICODE_TO_GBK[29747] := 16#CA75;
   // UNICODE_TO_GBK[29748] := 16#854D;
   // UNICODE_TO_GBK[29749] := 16#CA76;
   // UNICODE_TO_GBK[29750] := 16#854E;
   // UNICODE_TO_GBK[29751] := 16#CA77;
   // UNICODE_TO_GBK[29752] := 16#854F;
   // UNICODE_TO_GBK[29753] := 16#CA78;
   // UNICODE_TO_GBK[29754] := 16#8550;
   // UNICODE_TO_GBK[29755] := 16#CA79;
   // UNICODE_TO_GBK[29756] := 16#8551;
   // UNICODE_TO_GBK[29757] := 16#CA7A;
   // UNICODE_TO_GBK[29758] := 16#8552;
   // UNICODE_TO_GBK[29759] := 16#CA7B;
   // UNICODE_TO_GBK[29760] := 16#8553;
   // UNICODE_TO_GBK[29761] := 16#CA7C;
   // UNICODE_TO_GBK[29762] := 16#8554;
   // UNICODE_TO_GBK[29763] := 16#CA7D;
   // UNICODE_TO_GBK[29764] := 16#8555;
   // UNICODE_TO_GBK[29765] := 16#CA7E;
   // UNICODE_TO_GBK[29766] := 16#8556;
   // UNICODE_TO_GBK[29767] := 16#DEA1;
   // UNICODE_TO_GBK[29768] := 16#8557;
   // UNICODE_TO_GBK[29769] := 16#CA80;
   // UNICODE_TO_GBK[29770] := 16#8558;
   // UNICODE_TO_GBK[29771] := 16#CA81;
   // UNICODE_TO_GBK[29772] := 16#8559;
   // UNICODE_TO_GBK[29773] := 16#DEA5;
   // UNICODE_TO_GBK[29774] := 16#855A;
   // UNICODE_TO_GBK[29775] := 16#CA82;
   // UNICODE_TO_GBK[29776] := 16#855B;
   // UNICODE_TO_GBK[29777] := 16#CA83;
   // UNICODE_TO_GBK[29778] := 16#855C;
   // UNICODE_TO_GBK[29779] := 16#CA84;
   // UNICODE_TO_GBK[29780] := 16#855D;
   // UNICODE_TO_GBK[29781] := 16#CA85;
   // UNICODE_TO_GBK[29782] := 16#855E;
   // UNICODE_TO_GBK[29783] := 16#DEA9;
   // UNICODE_TO_GBK[29784] := 16#855F;
   // UNICODE_TO_GBK[29785] := 16#CA86;
   // UNICODE_TO_GBK[29786] := 16#8560;
   // UNICODE_TO_GBK[29787] := 16#CA87;
   // UNICODE_TO_GBK[29788] := 16#8561;
   // UNICODE_TO_GBK[29789] := 16#CA88;
   // UNICODE_TO_GBK[29790] := 16#8562;
   // UNICODE_TO_GBK[29791] := 16#CA89;
   // UNICODE_TO_GBK[29792] := 16#8563;
   // UNICODE_TO_GBK[29793] := 16#CA8A;
   // UNICODE_TO_GBK[29794] := 16#8564;
   // UNICODE_TO_GBK[29795] := 16#DEA8;
   // UNICODE_TO_GBK[29796] := 16#8565;
   // UNICODE_TO_GBK[29797] := 16#CA8B;
   // UNICODE_TO_GBK[29798] := 16#8566;
   // UNICODE_TO_GBK[29799] := 16#CA8C;
   // UNICODE_TO_GBK[29800] := 16#8567;
   // UNICODE_TO_GBK[29801] := 16#CA8D;
   // UNICODE_TO_GBK[29802] := 16#8568;
   // UNICODE_TO_GBK[29803] := 16#DEA7;
   // UNICODE_TO_GBK[29804] := 16#8569;
   // UNICODE_TO_GBK[29805] := 16#CA8E;
   // UNICODE_TO_GBK[29806] := 16#856A;
   // UNICODE_TO_GBK[29807] := 16#CA8F;
   // UNICODE_TO_GBK[29808] := 16#856B;
   // UNICODE_TO_GBK[29809] := 16#CA90;
   // UNICODE_TO_GBK[29810] := 16#856C;
   // UNICODE_TO_GBK[29811] := 16#CA91;
   // UNICODE_TO_GBK[29812] := 16#856D;
   // UNICODE_TO_GBK[29813] := 16#CA92;
   // UNICODE_TO_GBK[29814] := 16#856E;
   // UNICODE_TO_GBK[29815] := 16#CA93;
   // UNICODE_TO_GBK[29816] := 16#856F;
   // UNICODE_TO_GBK[29817] := 16#CA94;
   // UNICODE_TO_GBK[29818] := 16#8570;
   // UNICODE_TO_GBK[29819] := 16#CA95;
   // UNICODE_TO_GBK[29820] := 16#8571;
   // UNICODE_TO_GBK[29821] := 16#CA96;
   // UNICODE_TO_GBK[29822] := 16#8572;
   // UNICODE_TO_GBK[29823] := 16#DEAD;
   // UNICODE_TO_GBK[29824] := 16#8573;
   // UNICODE_TO_GBK[29825] := 16#CA97;
